// TIA Portal V20 export
FUNCTION_BLOCK "CallEquipment"   // FB177, LAD
TITLE = CallEquipment
// Template of an equipment module. This block contains the logic and futher calls (e.g. sequences, control modules, diagnostics etc.) of the equipment module.
// It can be used out of the box but also adapted to your own needs.
// stored: IsIECCheckEnabled true, MemoryReserve 100, Namespace Unit1.Em3, SetENOAutomatically true
   VAR_INPUT
      ZoneOperationEnable { ExternalWritable := 'False'} : "LWONIK_typeSafetyZoneManualOperation";
      unitEnableControlInterfaces { ExternalWritable := 'False'} : "LAF_typeEnableControlInterfaces";
      commandExcute { ExternalWritable := 'False'} : Bool;
   END_VAR
   VAR_IN_OUT
      unitStatus : "LAF_typeUnitStatus";   // Current unit status o be used in this EM
      emFeedback : "LUC_typeEmFeedback";   // Feedback of the EM to the Unit
      unitAlarmDB : "LAF_typeAlarms";   // Summarized EM Alarms for the Unit
   END_VAR
   VAR
      instSequenceWebGuid { ExternalWritable := 'False'} : "Unit1.Em3.Sequence_1_WebGuid";
      instWebGuidInitializedJob1 { ExternalWritable := 'False'} : "LAF_SelectJob";
      instWebGuidMotionCalculateJob2 { ExternalWritable := 'False'} : "LAF_SelectJob";
      instWebGuidMotionOneCellJob3 { ExternalWritable := 'False'} : "LAF_SelectJob";
      instWebGuidMotionFullStepJob4 { ExternalWritable := 'False'} : "LAF_SelectJob";
      instWebGuidMotionAutoJob5 { ExternalWritable := 'False'} : "LAF_SelectJob";
      instWebGuidMotionSemiStepJob6 { ExternalWritable := 'False'} : "LAF_SelectJob";
      instWebGuidMotionCycleStopJob7 { ExternalWritable := 'False'} : "LAF_SelectJob";
      instWebGuidMotionFastStopJob8 { ExternalWritable := 'False'} : "LAF_SelectJob";
      instCmMasterVirtualAxis { ExternalWritable := 'False'} : "LBC_AxisControl_TecPlcCn";
      instCmUnwinderVirtualAxis { ExternalWritable := 'False'} : "LBC_AxisControl_TecPlcCn";
      instCmDancerRegulatorOnOff { ExternalWritable := 'False'} : "LBC_TwoWayActuatorCn";
      instCmDancerSafetyPinIdlePosition { ExternalWritable := 'False'} : "LBC_DigitalSignalCn";
      instCmDancerEncoderAnalogInput { ExternalWritable := 'False'} : "LBC_AnalogInputCn";
      instCmLoadCellAnalogInput { ExternalWritable := 'False'} : "LBC_AnalogInputCn";
      instCmDancerElectroPneumaticRegulatorAnalogOutput { ExternalWritable := 'False'} : "LBC_AnalogOutputCn";
      instCmWebGuideEpc { ExternalWritable := 'False'} : "LER_EPC_CON600";
      instCmMasterAxisControlInterlockSummary { ExternalWritable := 'False'} : "LER_AxisControl_InterlockSummary";
      instCmUnwinderAxisControlInterlockSummary { ExternalWritable := 'False'} : "LER_AxisControl_InterlockSummary";
      statUnitStatus { ExternalWritable := 'False'} : "LAF_typeUnitStatus";   // Unit Status used in this EM
      instManageAlarms { ExternalWritable := 'False'} : "LAF_ManageAlarms";
      instEventsPFE { S7_SetPoint := 'True'} : "Unit1.Em3.EventsPFE";
      statLoadcellBuf { ExternalWritable := 'False'} : Int;
      statEnableManualCmds { ExternalWritable := 'False'} : Bool;
      statPulse { ExternalWritable := 'False'} : Array[0..99] of Bool;
      statTonTimer { ExternalWritable := 'False'} : Array[0..99] of TON_TIME;
      statTofTimer { ExternalWritable := 'False'} : Array[0..99] of TOF_TIME;
      instCheckCamRecipeChanged { ExternalWritable := 'False'} : "LER_CheckCamRecipeChanged";
      statCheckCamRecipeChangedStatus { ExternalWritable := 'False'} : Struct
         ValidParameters : Bool;
         ParameterChanged : Bool;
         ExecuteRequired : Bool;
      END_STRUCT;
      NGConveyorFull { ExternalVisible := 'False'; ExternalWritable := 'False'} : Bool;
      Stack1ConveyorFull { ExternalVisible := 'False'; ExternalWritable := 'False'} : Bool;
      Stack2ConveyorFull { ExternalVisible := 'False'; ExternalWritable := 'False'} : Bool;
      All_Full { ExternalVisible := 'False'; ExternalWritable := 'False'} : Bool;
      Stack1_Full_Abnormal { ExternalVisible := 'False'; ExternalWritable := 'False'} : Bool;
      Stack2_Full_Abnormal { ExternalVisible := 'False'; ExternalWritable := 'False'} : Bool;
      CutConveyorFull { ExternalVisible := 'False'; ExternalWritable := 'False'} : Bool;
      "Stack#1BA030Unuse" { ExternalVisible := 'False'; ExternalWritable := 'False'} : Bool;
      "Stack#2BA040Unuse" { ExternalVisible := 'False'; ExternalWritable := 'False'} : Bool;
      instCVFullChargeCheckCMD { S7_SetPoint := 'True'} : "LAF_SelectJob";
      CellCountDiv1 { S7_SetPoint := 'True'} : LReal;
      CellCountDiv2 { S7_SetPoint := 'True'} : LReal;
   END_VAR
   VAR_TEMP
      tempScInProduction : Bool;   // Mode Production and StateComplete
      tempScNoProduction : Bool;   // Mode Manual and StateComplete
   END_VAR
   VAR CONSTANT
      TO_DO_INSERT_PRECONDITIONS_HERE : Bool := TRUE;   // Template : Add em specific conditions here
      NO_JOB : DInt;   // No job
      TRUE : Bool := TRUE;
      FALSE : Bool := FALSE;
   END_VAR
   VAR_TEMP   // added for the SCL form of the ladder/FBD networks
      _w1 : Bool;
      _w2 : Bool;
   END_VAR
BEGIN

REGION Network 1: BLOCK INFO HEADER
   // (company) / (C) Copyright (year)
   // ---------------------------------------------------------------------------------
   // Title:                             (Title of this block)
   // Comment/Function: (that is implemented in the block)
   // Library/Family:           (that the source is dedicated to)
   // Author:                        (department / person in charge / contact)
   // Target System:          (test system with FW version)
   // Engineering:              TIA Portal (SW version)
   // Restrictions:               (OB types, etc.)
   // Requirements:           (hardware, technological package, etc.)
   // ---------------------------------------------------------------------------------
   // Change log table:
   // Version          | Date             | Signature      | Expert in charge  | Changes applied ------------------------|----------------------|-------------------------|--------------------------------|-----------------------
   // 001.000.000 | yyyy-mm-dd | 0x00000000 | (name of expert) | First released version
END_REGION

REGION Network 2: DESCRIPTION
   // This is a template block provided by the Automation Framework. It can be used to create an own project.
   // The Block Info Header is prepared to put in your own data.
   // Description of the block could be added here and the docu created by Code2Docu.
END_REGION

REGION Network 3: ******************** Equipment Control ********************
END_REGION

REGION Network 4: Interlink EM to Unit
   // This block links and unlinks the EM from the unit. The command to link/unlink can be set directly by the inputs of the block (e.g. to link/unlink based on any program logic) or through the InOut "hmiInterface". The block changes the output "isLinked" to true/false, depending on the command and if a change is allowed. A changed is allowed if the unit is in state aborted, clearing or stopped. The output "isLinked" is send back to the unit. If the EM is not linked, the unit ignores this EM.
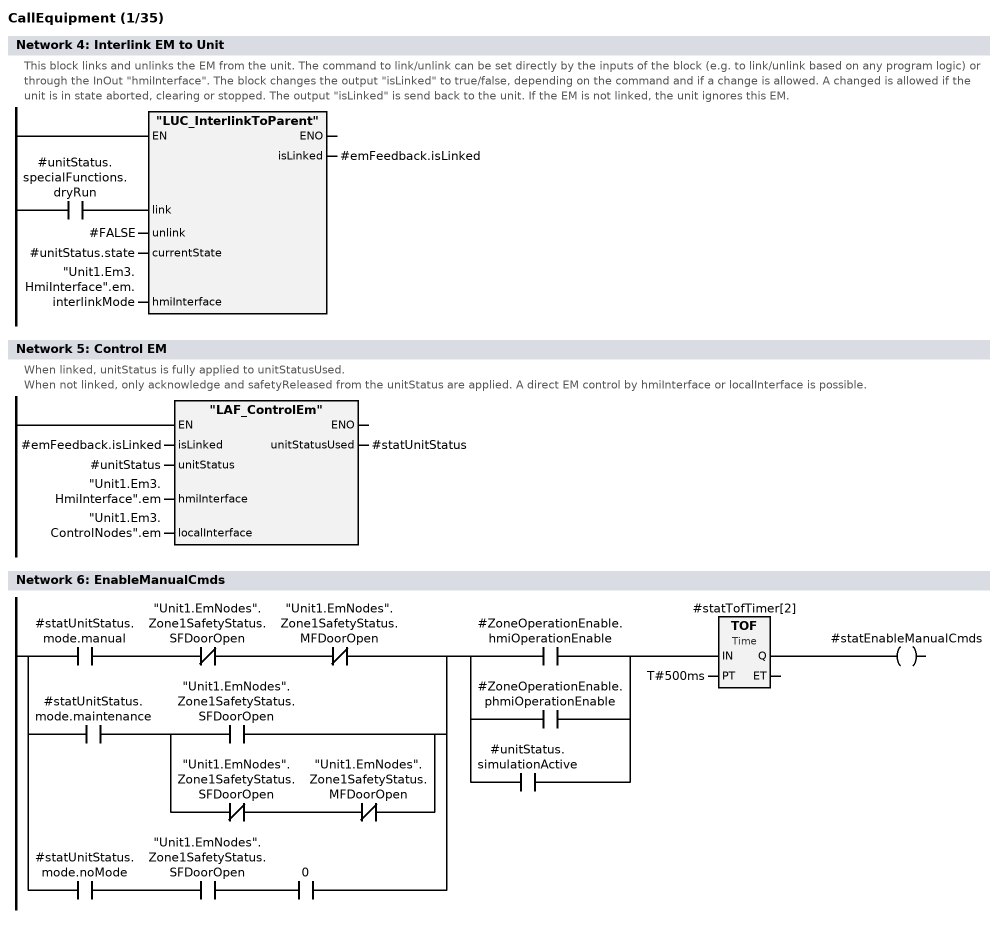
   RUNG wire#powerrail
      "LUC_InterlinkToParent"(link := wire#w1, unlink := #FALSE, currentState := #unitStatus.state, hmiInterface := "Unit1.Em3.HmiInterface".em.interlinkMode, isLinked => #emFeedback.isLinked)
   END_RUNG
   RUNG wire#powerrail
      Contact( #unitStatus.specialFunctions.dryRun )
   END_RUNG wire#w1
   // the same network as SCL:
   "LUC_InterlinkToParent"(link := #unitStatus.specialFunctions.dryRun,
                           unlink := #FALSE,
                           currentState := #unitStatus.state,
                           hmiInterface := "Unit1.Em3.HmiInterface".em.interlinkMode,
                           isLinked => #emFeedback.isLinked);
END_REGION

REGION Network 5: Control EM
   // When linked, unitStatus is fully applied to unitStatusUsed.
   // When not linked, only acknowledge and safetyReleased from the unitStatus are applied. A direct EM control by hmiInterface or localInterface is possible.
   RUNG wire#powerrail
      "LAF_ControlEm"(isLinked := #emFeedback.isLinked, unitStatus := #unitStatus, hmiInterface := "Unit1.Em3.HmiInterface".em, localInterface := "Unit1.Em3.ControlNodes".em, unitStatusUsed => #statUnitStatus)
   END_RUNG
   // the same network as SCL:
   "LAF_ControlEm"(isLinked := #emFeedback.isLinked,
                   unitStatus := #unitStatus,
                   hmiInterface := "Unit1.Em3.HmiInterface".em,
                   localInterface := "Unit1.Em3.ControlNodes".em,
                   unitStatusUsed => #statUnitStatus);
END_REGION

REGION Network 6: EnableManualCmds
   RUNG wire#powerrail
      Contact( #statUnitStatus.mode.manual )
      I_Contact( "Unit1.EmNodes".Zone1SafetyStatus.SFDoorOpen )
      I_Contact( "Unit1.EmNodes".Zone1SafetyStatus.MFDoorOpen )
      wire#w1
      Contact( #ZoneOperationEnable.hmiOperationEnable )
      wire#w3
      { S7_Templates := "time_type := Time" } #statTofTimer[2].TOF(pt := T#500ms, et =>)
      Coil( #statEnableManualCmds )
   END_RUNG
   RUNG wire#powerrail
      Contact( #statUnitStatus.mode.maintenance )
      wire#w2
      Contact( "Unit1.EmNodes".Zone1SafetyStatus.SFDoorOpen )
   END_RUNG wire#w1
   RUNG wire#w2
      I_Contact( "Unit1.EmNodes".Zone1SafetyStatus.SFDoorOpen )
      I_Contact( "Unit1.EmNodes".Zone1SafetyStatus.MFDoorOpen )
   END_RUNG wire#w1
   RUNG wire#powerrail
      Contact( #statUnitStatus.mode.noMode )
      Contact( "Unit1.EmNodes".Zone1SafetyStatus.SFDoorOpen )
      Contact( 0 )
   END_RUNG wire#w1
   RUNG wire#w1
      Contact( #ZoneOperationEnable.phmiOperationEnable )
   END_RUNG wire#w3
   RUNG wire#w1
      Contact( #unitStatus.simulationActive )
   END_RUNG wire#w3
   // the same network as SCL:
   #statTofTimer[2].TOF(IN := ((#statUnitStatus.mode.manual AND NOT "Unit1.EmNodes".Zone1SafetyStatus.SFDoorOpen AND NOT "Unit1.EmNodes".Zone1SafetyStatus.MFDoorOpen) OR (#statUnitStatus.mode.maintenance AND ("Unit1.EmNodes".Zone1SafetyStatus.SFDoorOpen OR (NOT "Unit1.EmNodes".Zone1SafetyStatus.SFDoorOpen AND NOT "Unit1.EmNodes".Zone1SafetyStatus.MFDoorOpen))) OR (#statUnitStatus.mode.noMode AND "Unit1.EmNodes".Zone1SafetyStatus.SFDoorOpen AND 0)) AND (#ZoneOperationEnable.hmiOperationEnable OR #ZoneOperationEnable.phmiOperationEnable OR #unitStatus.simulationActive),
                        PT := T#500ms);
   #statEnableManualCmds := #statTofTimer[2].Q;
END_REGION

REGION Network 7: Alarms Disabled
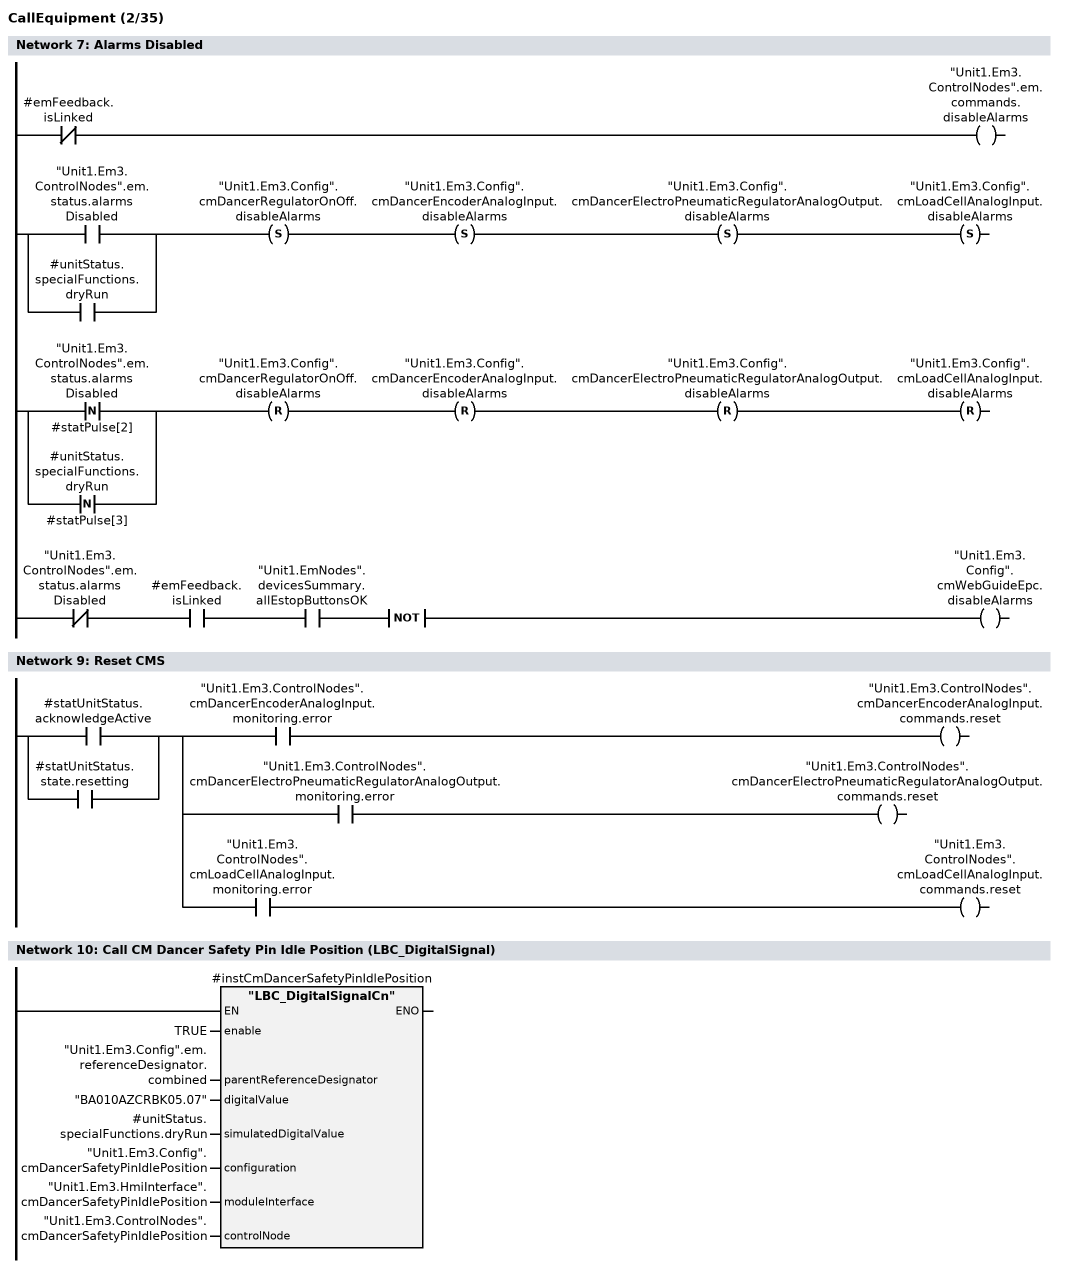
   RUNG wire#powerrail
      I_Contact( #emFeedback.isLinked )
      Coil( "Unit1.Em3.ControlNodes".em.commands.disableAlarms )
   END_RUNG
   RUNG wire#powerrail
      Contact( "Unit1.Em3.ControlNodes".em.status.alarmsDisabled )
      wire#w1
      S_Coil( "Unit1.Em3.Config".cmDancerRegulatorOnOff.disableAlarms )
      S_Coil( "Unit1.Em3.Config".cmDancerEncoderAnalogInput.disableAlarms )
      S_Coil( "Unit1.Em3.Config".cmDancerElectroPneumaticRegulatorAnalogOutput.disableAlarms )
      S_Coil( "Unit1.Em3.Config".cmLoadCellAnalogInput.disableAlarms )
   END_RUNG
   RUNG wire#powerrail
      Contact( #unitStatus.specialFunctions.dryRun )
   END_RUNG wire#w1
   RUNG wire#powerrail
      N_Contact(operand := "Unit1.Em3.ControlNodes".em.status.alarmsDisabled, bit := #statPulse[2])
      wire#w2
      R_Coil( "Unit1.Em3.Config".cmDancerRegulatorOnOff.disableAlarms )
      R_Coil( "Unit1.Em3.Config".cmDancerEncoderAnalogInput.disableAlarms )
      R_Coil( "Unit1.Em3.Config".cmDancerElectroPneumaticRegulatorAnalogOutput.disableAlarms )
      R_Coil( "Unit1.Em3.Config".cmLoadCellAnalogInput.disableAlarms )
   END_RUNG
   RUNG wire#powerrail
      N_Contact(operand := #unitStatus.specialFunctions.dryRun, bit := #statPulse[3])
   END_RUNG wire#w2
   RUNG wire#powerrail
      I_Contact( "Unit1.Em3.ControlNodes".em.status.alarmsDisabled )
      Contact( #emFeedback.isLinked )
      Contact( "Unit1.EmNodes".devicesSummary.allEstopButtonsOK )
      Not()
      Coil( "Unit1.Em3.Config".cmWebGuideEpc.disableAlarms )
   END_RUNG
   // the same network as SCL:
   "Unit1.Em3.ControlNodes".em.commands.disableAlarms := NOT #emFeedback.isLinked;
   IF "Unit1.Em3.ControlNodes".em.status.alarmsDisabled OR #unitStatus.specialFunctions.dryRun THEN
       "Unit1.Em3.Config".cmDancerRegulatorOnOff.disableAlarms := TRUE;
       "Unit1.Em3.Config".cmDancerEncoderAnalogInput.disableAlarms := TRUE;
       "Unit1.Em3.Config".cmDancerElectroPneumaticRegulatorAnalogOutput.disableAlarms := TRUE;
       "Unit1.Em3.Config".cmLoadCellAnalogInput.disableAlarms := TRUE;
   END_IF;
   #_w1 := NOT "Unit1.Em3.ControlNodes".em.status.alarmsDisabled AND #statPulse[2];   // falling edge of "Unit1.Em3.ControlNodes".em.status.alarmsDisabled
   #statPulse[2] := "Unit1.Em3.ControlNodes".em.status.alarmsDisabled;
   #_w2 := NOT #unitStatus.specialFunctions.dryRun AND #statPulse[3];   // falling edge of #unitStatus.specialFunctions.dryRun
   #statPulse[3] := #unitStatus.specialFunctions.dryRun;
   IF #_w1 OR #_w2 THEN
       "Unit1.Em3.Config".cmDancerRegulatorOnOff.disableAlarms := FALSE;
       "Unit1.Em3.Config".cmDancerEncoderAnalogInput.disableAlarms := FALSE;
       "Unit1.Em3.Config".cmDancerElectroPneumaticRegulatorAnalogOutput.disableAlarms := FALSE;
       "Unit1.Em3.Config".cmLoadCellAnalogInput.disableAlarms := FALSE;
   END_IF;
   "Unit1.Em3.Config".cmWebGuideEpc.disableAlarms := NOT (NOT "Unit1.Em3.ControlNodes".em.status.alarmsDisabled AND #emFeedback.isLinked AND "Unit1.EmNodes".devicesSummary.allEstopButtonsOK);
END_REGION

REGION Network 8: ******************** Control Modules (Sensors) ********************
   // Call control modules that are sensors before the em logic (jobs and sequence), so that the latest value is used in the logic.
END_REGION

REGION Network 9: Reset CMS
   RUNG wire#powerrail
      Contact( #statUnitStatus.acknowledgeActive )
      wire#w1
      Contact( "Unit1.Em3.ControlNodes".cmDancerEncoderAnalogInput.monitoring.error )
      Coil( "Unit1.Em3.ControlNodes".cmDancerEncoderAnalogInput.commands.reset )
   END_RUNG
   RUNG wire#powerrail
      Contact( #statUnitStatus.state.resetting )
   END_RUNG wire#w1
   RUNG wire#w1
      Contact( "Unit1.Em3.ControlNodes".cmDancerElectroPneumaticRegulatorAnalogOutput.monitoring.error )
      Coil( "Unit1.Em3.ControlNodes".cmDancerElectroPneumaticRegulatorAnalogOutput.commands.reset )
   END_RUNG
   RUNG wire#w1
      Contact( "Unit1.Em3.ControlNodes".cmLoadCellAnalogInput.monitoring.error )
      Coil( "Unit1.Em3.ControlNodes".cmLoadCellAnalogInput.commands.reset )
   END_RUNG
   // the same network as SCL:
   #_w1 := #statUnitStatus.acknowledgeActive OR #statUnitStatus.state.resetting;
   "Unit1.Em3.ControlNodes".cmDancerEncoderAnalogInput.commands.reset := #_w1 AND "Unit1.Em3.ControlNodes".cmDancerEncoderAnalogInput.monitoring.error;
   "Unit1.Em3.ControlNodes".cmDancerElectroPneumaticRegulatorAnalogOutput.commands.reset := #_w1 AND "Unit1.Em3.ControlNodes".cmDancerElectroPneumaticRegulatorAnalogOutput.monitoring.error;
   "Unit1.Em3.ControlNodes".cmLoadCellAnalogInput.commands.reset := #_w1 AND "Unit1.Em3.ControlNodes".cmLoadCellAnalogInput.monitoring.error;
END_REGION

REGION Network 10: Call CM Dancer Safety Pin Idle Position (LBC_DigitalSignal)
   RUNG wire#powerrail
      #instCmDancerSafetyPinIdlePosition(enable := TRUE, parentReferenceDesignator := "Unit1.Em3.Config".em.referenceDesignator.combined, digitalValue := "BA010AZCRBK05.07", simulatedDigitalValue := #unitStatus.specialFunctions.dryRun, configuration := "Unit1.Em3.Config".cmDancerSafetyPinIdlePosition, moduleInterface := "Unit1.Em3.HmiInterface".cmDancerSafetyPinIdlePosition, controlNode := "Unit1.Em3.ControlNodes".cmDancerSafetyPinIdlePosition)
   END_RUNG
   // the same network as SCL:
   #instCmDancerSafetyPinIdlePosition(enable := TRUE,   // "LBC_DigitalSignalCn"
                           parentReferenceDesignator := "Unit1.Em3.Config".em.referenceDesignator.combined,
                           digitalValue := "BA010AZCRBK05.07",
                           simulatedDigitalValue := #unitStatus.specialFunctions.dryRun,
                           configuration := "Unit1.Em3.Config".cmDancerSafetyPinIdlePosition,
                           moduleInterface := "Unit1.Em3.HmiInterface".cmDancerSafetyPinIdlePosition,
                           controlNode := "Unit1.Em3.ControlNodes".cmDancerSafetyPinIdlePosition);
END_REGION

REGION Network 11: Call CM Load Cell (LBC_AnalogInput)
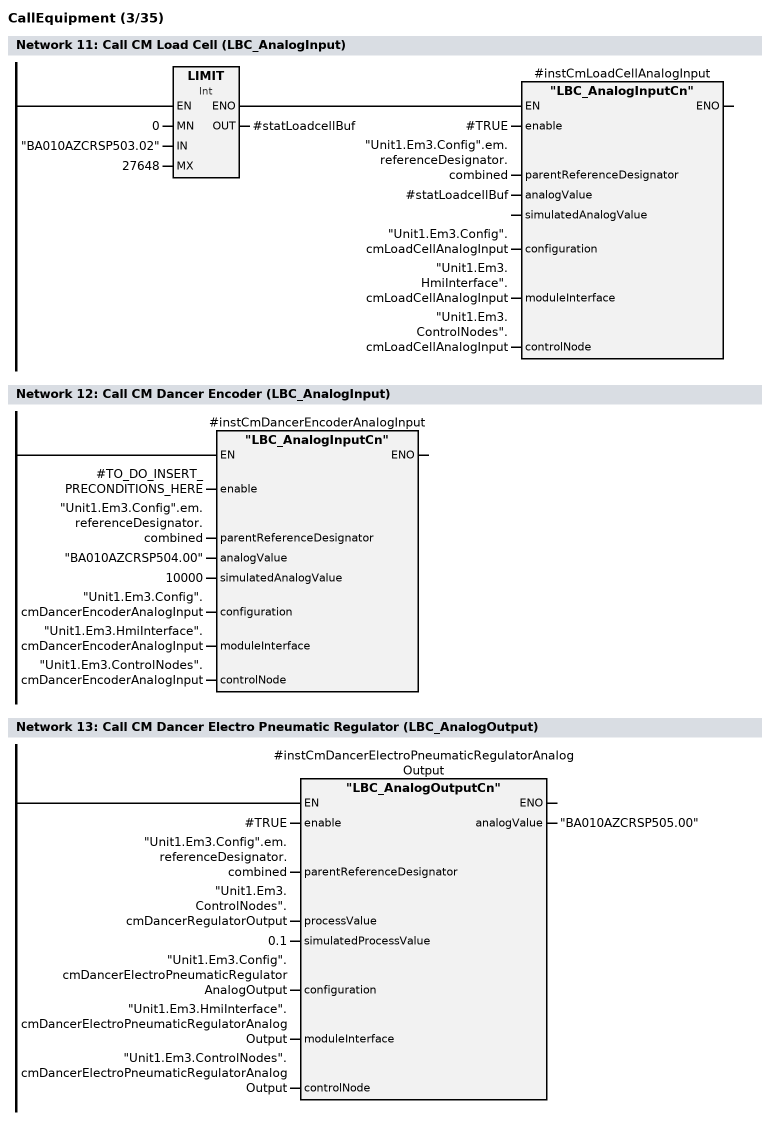
   RUNG wire#powerrail
      { S7_Templates := "value_type := Int" } Limit(mn := 0, in := "BA010AZCRSP503.02", mx := 27648, out => #statLoadcellBuf)
      #instCmLoadCellAnalogInput(enable := #TRUE, parentReferenceDesignator := "Unit1.Em3.Config".em.referenceDesignator.combined, analogValue := #statLoadcellBuf, simulatedAnalogValue :=, configuration := "Unit1.Em3.Config".cmLoadCellAnalogInput, moduleInterface := "Unit1.Em3.HmiInterface".cmLoadCellAnalogInput, controlNode := "Unit1.Em3.ControlNodes".cmLoadCellAnalogInput)
   END_RUNG
   // the same network as SCL:
   #statLoadcellBuf := LIMIT(MN := 0, IN := "BA010AZCRSP503.02", MX := 27648);
   #instCmLoadCellAnalogInput(enable := #TRUE,   // "LBC_AnalogInputCn"
                           parentReferenceDesignator := "Unit1.Em3.Config".em.referenceDesignator.combined,
                           analogValue := #statLoadcellBuf,
                           configuration := "Unit1.Em3.Config".cmLoadCellAnalogInput,
                           moduleInterface := "Unit1.Em3.HmiInterface".cmLoadCellAnalogInput,
                           controlNode := "Unit1.Em3.ControlNodes".cmLoadCellAnalogInput);
END_REGION

REGION Network 12: Call CM Dancer Encoder (LBC_AnalogInput)
   RUNG wire#powerrail
      #instCmDancerEncoderAnalogInput(enable := #TO_DO_INSERT_PRECONDITIONS_HERE, parentReferenceDesignator := "Unit1.Em3.Config".em.referenceDesignator.combined, analogValue := "BA010AZCRSP504.00", simulatedAnalogValue := 10000, configuration := "Unit1.Em3.Config".cmDancerEncoderAnalogInput, moduleInterface := "Unit1.Em3.HmiInterface".cmDancerEncoderAnalogInput, controlNode := "Unit1.Em3.ControlNodes".cmDancerEncoderAnalogInput)
   END_RUNG
   // the same network as SCL:
   #instCmDancerEncoderAnalogInput(enable := #TO_DO_INSERT_PRECONDITIONS_HERE,   // "LBC_AnalogInputCn"
                           parentReferenceDesignator := "Unit1.Em3.Config".em.referenceDesignator.combined,
                           analogValue := "BA010AZCRSP504.00",
                           simulatedAnalogValue := 10000,
                           configuration := "Unit1.Em3.Config".cmDancerEncoderAnalogInput,
                           moduleInterface := "Unit1.Em3.HmiInterface".cmDancerEncoderAnalogInput,
                           controlNode := "Unit1.Em3.ControlNodes".cmDancerEncoderAnalogInput);
END_REGION

REGION Network 13: Call CM Dancer Electro Pneumatic Regulator (LBC_AnalogOutput)
   RUNG wire#powerrail
      #instCmDancerElectroPneumaticRegulatorAnalogOutput(enable := #TRUE, parentReferenceDesignator := "Unit1.Em3.Config".em.referenceDesignator.combined, processValue := "Unit1.Em3.ControlNodes".cmDancerRegulatorOutput, simulatedProcessValue := 0.1, configuration := "Unit1.Em3.Config".cmDancerElectroPneumaticRegulatorAnalogOutput, moduleInterface := "Unit1.Em3.HmiInterface".cmDancerElectroPneumaticRegulatorAnalogOutput, controlNode := "Unit1.Em3.ControlNodes".cmDancerElectroPneumaticRegulatorAnalogOutput, analogValue => "BA010AZCRSP505.00")
   END_RUNG
   // the same network as SCL:
   #instCmDancerElectroPneumaticRegulatorAnalogOutput(enable := #TRUE,   // "LBC_AnalogOutputCn"
                           parentReferenceDesignator := "Unit1.Em3.Config".em.referenceDesignator.combined,
                           processValue := "Unit1.Em3.ControlNodes".cmDancerRegulatorOutput,
                           simulatedProcessValue := 0.1,
                           configuration := "Unit1.Em3.Config".cmDancerElectroPneumaticRegulatorAnalogOutput,
                           moduleInterface := "Unit1.Em3.HmiInterface".cmDancerElectroPneumaticRegulatorAnalogOutput,
                           controlNode := "Unit1.Em3.ControlNodes".cmDancerElectroPneumaticRegulatorAnalogOutput,
                           analogValue => "BA010AZCRSP505.00");
END_REGION

REGION Network 14: ******************** Equipment Logic ********************
END_REGION

REGION Network 15: Map Unit Status to Sequence Status [1] WebGuid
   // This block maps the unit status to the seuqnce status. Thus, it controls the sequence depending on the unit status. E.g. it sets the sequence to automatic when the unit state is in productions. This blocks work perfectly with the sequences provided in the AF. 
   // This typed block (MapUnitStatusToSequence) could be adjusted to specific application requirements or if other, user-defined sequences are used.
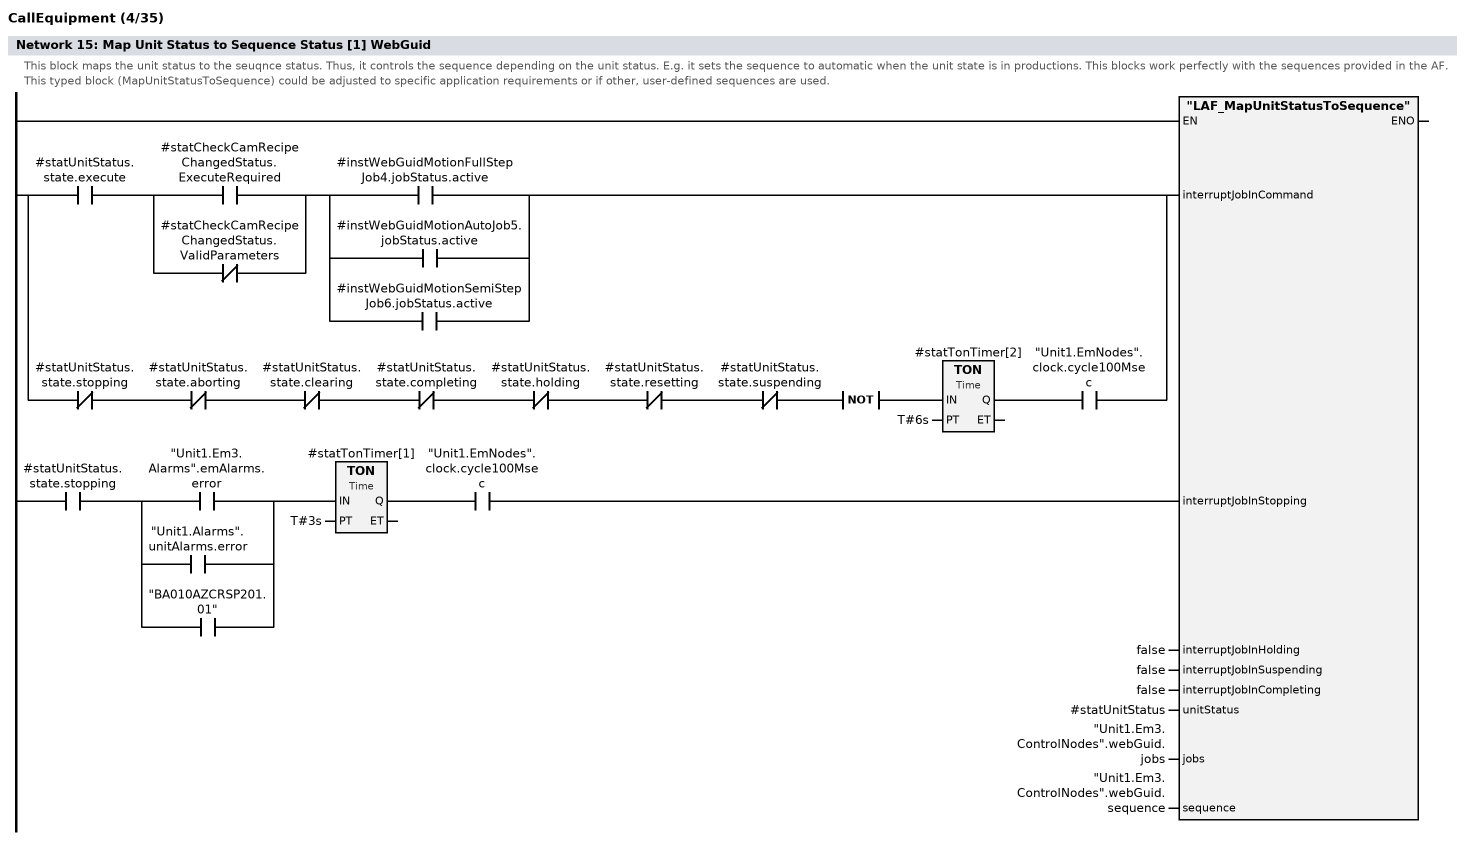
   RUNG wire#powerrail
      "LAF_MapUnitStatusToSequence"(interruptJobInCommand := wire#w3, interruptJobInStopping := wire#w6, interruptJobInHolding := false, interruptJobInSuspending := false, interruptJobInCompleting := false, unitStatus := #statUnitStatus, jobs := "Unit1.Em3.ControlNodes".webGuid.jobs, sequence := "Unit1.Em3.ControlNodes".webGuid.sequence)
   END_RUNG
   RUNG wire#powerrail
      Contact( #statUnitStatus.state.execute )
      wire#w1
      Contact( #statCheckCamRecipeChangedStatus.ExecuteRequired )
      wire#w2
      Contact( #instWebGuidMotionFullStepJob4.jobStatus.active )
   END_RUNG wire#w3
   RUNG wire#w1
      I_Contact( #statCheckCamRecipeChangedStatus.ValidParameters )
   END_RUNG wire#w2
   RUNG wire#w2
      Contact( #instWebGuidMotionAutoJob5.jobStatus.active )
   END_RUNG wire#w3
   RUNG wire#w2
      Contact( #instWebGuidMotionSemiStepJob6.jobStatus.active )
   END_RUNG wire#w3
   RUNG wire#powerrail
      I_Contact( #statUnitStatus.state.stopping )
      I_Contact( #statUnitStatus.state.aborting )
      I_Contact( #statUnitStatus.state.clearing )
      I_Contact( #statUnitStatus.state.completing )
      I_Contact( #statUnitStatus.state.holding )
      I_Contact( #statUnitStatus.state.resetting )
      I_Contact( #statUnitStatus.state.suspending )
      Not()
      { S7_Templates := "time_type := Time" } #statTonTimer[2].TON(pt := T#6s, et =>)
      Contact( "Unit1.EmNodes".clock.cycle100Msec )
   END_RUNG wire#w3
   RUNG wire#powerrail
      Contact( #statUnitStatus.state.stopping )
      wire#w4
      Contact( "Unit1.Em3.Alarms".emAlarms.error )
      wire#w5
      { S7_Templates := "time_type := Time" } #statTonTimer[1].TON(pt := T#3s, et =>)
      Contact( "Unit1.EmNodes".clock.cycle100Msec )
   END_RUNG wire#w6
   RUNG wire#w4
      Contact( "Unit1.Alarms".unitAlarms.error )
   END_RUNG wire#w5
   RUNG wire#w4
      Contact( "BA010AZCRSP201.01" )
   END_RUNG wire#w5
   // the same network as SCL:
   #statTonTimer[2].TON(IN := NOT (NOT #statUnitStatus.state.stopping AND NOT #statUnitStatus.state.aborting AND NOT #statUnitStatus.state.clearing AND NOT #statUnitStatus.state.completing AND NOT #statUnitStatus.state.holding AND NOT #statUnitStatus.state.resetting AND NOT #statUnitStatus.state.suspending),
                        PT := T#6s);
   #_w1 := (#statUnitStatus.state.execute AND (#statCheckCamRecipeChangedStatus.ExecuteRequired OR NOT #statCheckCamRecipeChangedStatus.ValidParameters) AND (#instWebGuidMotionFullStepJob4.jobStatus.active OR #instWebGuidMotionAutoJob5.jobStatus.active OR #instWebGuidMotionSemiStepJob6.jobStatus.active)) OR (#statTonTimer[2].Q AND "Unit1.EmNodes".clock.cycle100Msec);
   #statTonTimer[1].TON(IN := #statUnitStatus.state.stopping AND ("Unit1.Em3.Alarms".emAlarms.error OR "Unit1.Alarms".unitAlarms.error OR "BA010AZCRSP201.01"),
                        PT := T#3s);
   "LAF_MapUnitStatusToSequence"(interruptJobInCommand := #_w1,
                           interruptJobInStopping := #statTonTimer[1].Q AND "Unit1.EmNodes".clock.cycle100Msec,
                           interruptJobInHolding := false,
                           interruptJobInSuspending := false,
                           interruptJobInCompleting := false,
                           unitStatus := #statUnitStatus,
                           jobs := "Unit1.Em3.ControlNodes".webGuid.jobs,
                           sequence := "Unit1.Em3.ControlNodes".webGuid.sequence);
END_REGION

REGION Network 16: C/V Full Charge Check before motion job select
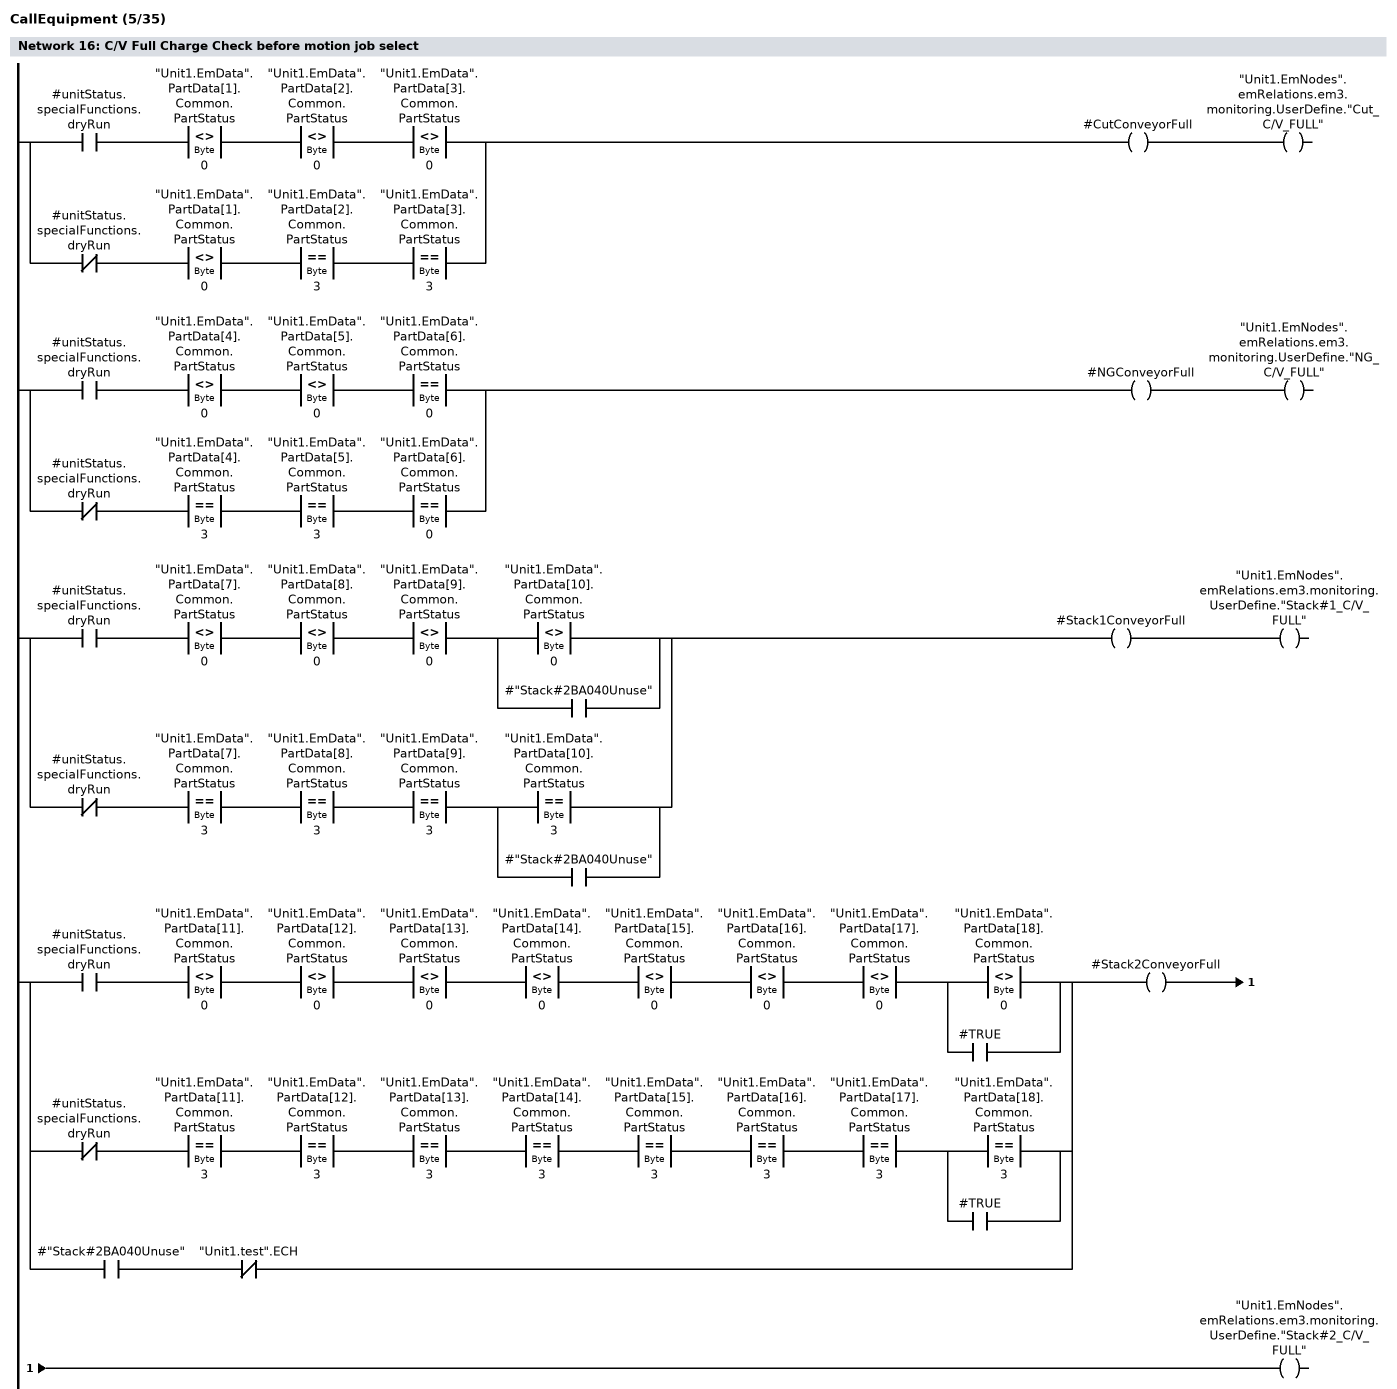
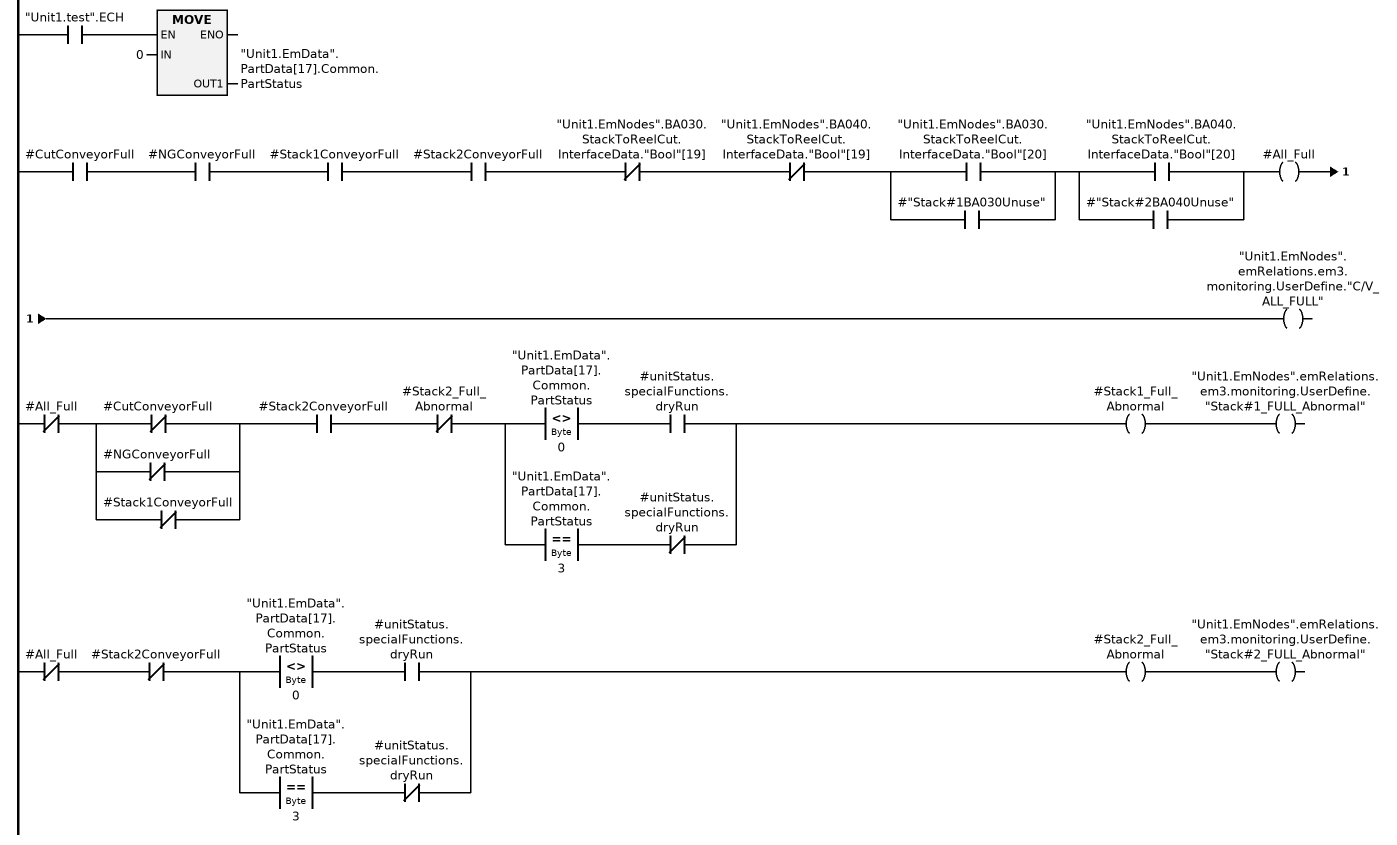
   RUNG wire#powerrail
      Contact( #unitStatus.specialFunctions.dryRun )
      { S7_Templates := "SrcType := Byte" } NE_Contact(in1 := "Unit1.EmData".PartData[1].Common.PartStatus, in2 := 0)
      { S7_Templates := "SrcType := Byte" } NE_Contact(in1 := "Unit1.EmData".PartData[2].Common.PartStatus, in2 := 0)
      { S7_Templates := "SrcType := Byte" } NE_Contact(in1 := "Unit1.EmData".PartData[3].Common.PartStatus, in2 := 0)
      wire#w1
      Coil( #CutConveyorFull )
      Coil( "Unit1.EmNodes".emRelations.em3.monitoring.UserDefine."Cut_C/V_FULL" )
   END_RUNG
   RUNG wire#powerrail
      I_Contact( #unitStatus.specialFunctions.dryRun )
      { S7_Templates := "SrcType := Byte" } NE_Contact(in1 := "Unit1.EmData".PartData[1].Common.PartStatus, in2 := 0)
      { S7_Templates := "SrcType := Byte" } EQ_Contact(in1 := "Unit1.EmData".PartData[2].Common.PartStatus, in2 := 3)
      { S7_Templates := "SrcType := Byte" } EQ_Contact(in1 := "Unit1.EmData".PartData[3].Common.PartStatus, in2 := 3)
   END_RUNG wire#w1
   RUNG wire#powerrail
      Contact( #unitStatus.specialFunctions.dryRun )
      { S7_Templates := "SrcType := Byte" } NE_Contact(in1 := "Unit1.EmData".PartData[4].Common.PartStatus, in2 := 0)
      { S7_Templates := "SrcType := Byte" } NE_Contact(in1 := "Unit1.EmData".PartData[5].Common.PartStatus, in2 := 0)
      { S7_Templates := "SrcType := Byte" } EQ_Contact(in1 := "Unit1.EmData".PartData[6].Common.PartStatus, in2 := 0)
      wire#w2
      Coil( #NGConveyorFull )
      Coil( "Unit1.EmNodes".emRelations.em3.monitoring.UserDefine."NG_C/V_FULL" )
   END_RUNG
   RUNG wire#powerrail
      I_Contact( #unitStatus.specialFunctions.dryRun )
      { S7_Templates := "SrcType := Byte" } EQ_Contact(in1 := "Unit1.EmData".PartData[4].Common.PartStatus, in2 := 3)
      { S7_Templates := "SrcType := Byte" } EQ_Contact(in1 := "Unit1.EmData".PartData[5].Common.PartStatus, in2 := 3)
      { S7_Templates := "SrcType := Byte" } EQ_Contact(in1 := "Unit1.EmData".PartData[6].Common.PartStatus, in2 := 0)
   END_RUNG wire#w2
   RUNG wire#powerrail
      Contact( #unitStatus.specialFunctions.dryRun )
      { S7_Templates := "SrcType := Byte" } NE_Contact(in1 := "Unit1.EmData".PartData[7].Common.PartStatus, in2 := 0)
      { S7_Templates := "SrcType := Byte" } NE_Contact(in1 := "Unit1.EmData".PartData[8].Common.PartStatus, in2 := 0)
      { S7_Templates := "SrcType := Byte" } NE_Contact(in1 := "Unit1.EmData".PartData[9].Common.PartStatus, in2 := 0)
      wire#w3
      { S7_Templates := "SrcType := Byte" } NE_Contact(in1 := "Unit1.EmData".PartData[10].Common.PartStatus, in2 := 0)
      wire#w4
      Coil( #Stack1ConveyorFull )
      Coil( "Unit1.EmNodes".emRelations.em3.monitoring.UserDefine."Stack#1_C/V_FULL" )
   END_RUNG
   RUNG wire#w3
      Contact( #"Stack#2BA040Unuse" )
   END_RUNG wire#w4
   RUNG wire#powerrail
      I_Contact( #unitStatus.specialFunctions.dryRun )
      { S7_Templates := "SrcType := Byte" } EQ_Contact(in1 := "Unit1.EmData".PartData[7].Common.PartStatus, in2 := 3)
      { S7_Templates := "SrcType := Byte" } EQ_Contact(in1 := "Unit1.EmData".PartData[8].Common.PartStatus, in2 := 3)
      { S7_Templates := "SrcType := Byte" } EQ_Contact(in1 := "Unit1.EmData".PartData[9].Common.PartStatus, in2 := 3)
      wire#w5
      { S7_Templates := "SrcType := Byte" } EQ_Contact(in1 := "Unit1.EmData".PartData[10].Common.PartStatus, in2 := 3)
   END_RUNG wire#w4
   RUNG wire#w5
      Contact( #"Stack#2BA040Unuse" )
   END_RUNG wire#w4
   RUNG wire#powerrail
      Contact( #unitStatus.specialFunctions.dryRun )
      { S7_Templates := "SrcType := Byte" } NE_Contact(in1 := "Unit1.EmData".PartData[11].Common.PartStatus, in2 := 0)
      { S7_Templates := "SrcType := Byte" } NE_Contact(in1 := "Unit1.EmData".PartData[12].Common.PartStatus, in2 := 0)
      { S7_Templates := "SrcType := Byte" } NE_Contact(in1 := "Unit1.EmData".PartData[13].Common.PartStatus, in2 := 0)
      { S7_Templates := "SrcType := Byte" } NE_Contact(in1 := "Unit1.EmData".PartData[14].Common.PartStatus, in2 := 0)
      { S7_Templates := "SrcType := Byte" } NE_Contact(in1 := "Unit1.EmData".PartData[15].Common.PartStatus, in2 := 0)
      { S7_Templates := "SrcType := Byte" } NE_Contact(in1 := "Unit1.EmData".PartData[16].Common.PartStatus, in2 := 0)
      { S7_Templates := "SrcType := Byte" } NE_Contact(in1 := "Unit1.EmData".PartData[17].Common.PartStatus, in2 := 0)
      wire#w6
      { S7_Templates := "SrcType := Byte" } NE_Contact(in1 := "Unit1.EmData".PartData[18].Common.PartStatus, in2 := 0)
      wire#w7
      Coil( #Stack2ConveyorFull )
      Coil( "Unit1.EmNodes".emRelations.em3.monitoring.UserDefine."Stack#2_C/V_FULL" )
   END_RUNG
   RUNG wire#w6
      Contact( #TRUE )
   END_RUNG wire#w7
   RUNG wire#powerrail
      I_Contact( #unitStatus.specialFunctions.dryRun )
      { S7_Templates := "SrcType := Byte" } EQ_Contact(in1 := "Unit1.EmData".PartData[11].Common.PartStatus, in2 := 3)
      { S7_Templates := "SrcType := Byte" } EQ_Contact(in1 := "Unit1.EmData".PartData[12].Common.PartStatus, in2 := 3)
      { S7_Templates := "SrcType := Byte" } EQ_Contact(in1 := "Unit1.EmData".PartData[13].Common.PartStatus, in2 := 3)
      { S7_Templates := "SrcType := Byte" } EQ_Contact(in1 := "Unit1.EmData".PartData[14].Common.PartStatus, in2 := 3)
      { S7_Templates := "SrcType := Byte" } EQ_Contact(in1 := "Unit1.EmData".PartData[15].Common.PartStatus, in2 := 3)
      { S7_Templates := "SrcType := Byte" } EQ_Contact(in1 := "Unit1.EmData".PartData[16].Common.PartStatus, in2 := 3)
      { S7_Templates := "SrcType := Byte" } EQ_Contact(in1 := "Unit1.EmData".PartData[17].Common.PartStatus, in2 := 3)
      wire#w8
      { S7_Templates := "SrcType := Byte" } EQ_Contact(in1 := "Unit1.EmData".PartData[18].Common.PartStatus, in2 := 3)
   END_RUNG wire#w7
   RUNG wire#w8
      Contact( #TRUE )
   END_RUNG wire#w7
   RUNG wire#powerrail
      Contact( #"Stack#2BA040Unuse" )
      I_Contact( "Unit1.test".ECH )
   END_RUNG wire#w7
   RUNG wire#powerrail
      Contact( "Unit1.test".ECH )
      Move(in := 0, out1 => "Unit1.EmData".PartData[17].Common.PartStatus)
   END_RUNG
   RUNG wire#powerrail
      Contact( #CutConveyorFull )
      Contact( #NGConveyorFull )
      Contact( #Stack1ConveyorFull )
      Contact( #Stack2ConveyorFull )
      I_Contact( "Unit1.EmNodes".BA030.StackToReelCut.InterfaceData."Bool"[19] )
      I_Contact( "Unit1.EmNodes".BA040.StackToReelCut.InterfaceData."Bool"[19] )
      wire#w9
      Contact( "Unit1.EmNodes".BA030.StackToReelCut.InterfaceData."Bool"[20] )
      wire#w10
      Contact( "Unit1.EmNodes".BA040.StackToReelCut.InterfaceData."Bool"[20] )
      wire#w11
      Coil( #All_Full )
      Coil( "Unit1.EmNodes".emRelations.em3.monitoring.UserDefine."C/V_ALL_FULL" )
   END_RUNG
   RUNG wire#w9
      Contact( #"Stack#1BA030Unuse" )
   END_RUNG wire#w10
   RUNG wire#w10
      Contact( #"Stack#2BA040Unuse" )
   END_RUNG wire#w11
   RUNG wire#powerrail
      I_Contact( #All_Full )
      wire#w12
      I_Contact( #CutConveyorFull )
      wire#w13
      Contact( #Stack2ConveyorFull )
      I_Contact( #Stack2_Full_Abnormal )
      wire#w14
      { S7_Templates := "SrcType := Byte" } NE_Contact(in1 := "Unit1.EmData".PartData[17].Common.PartStatus, in2 := 0)
      Contact( #unitStatus.specialFunctions.dryRun )
      wire#w15
      Coil( #Stack1_Full_Abnormal )
      Coil( "Unit1.EmNodes".emRelations.em3.monitoring.UserDefine."Stack#1_FULL_Abnormal" )
   END_RUNG
   RUNG wire#w12
      I_Contact( #NGConveyorFull )
   END_RUNG wire#w13
   RUNG wire#w12
      I_Contact( #Stack1ConveyorFull )
   END_RUNG wire#w13
   RUNG wire#w14
      { S7_Templates := "SrcType := Byte" } EQ_Contact(in1 := "Unit1.EmData".PartData[17].Common.PartStatus, in2 := 3)
      I_Contact( #unitStatus.specialFunctions.dryRun )
   END_RUNG wire#w15
   RUNG wire#powerrail
      I_Contact( #All_Full )
      I_Contact( #Stack2ConveyorFull )
      wire#w16
      { S7_Templates := "SrcType := Byte" } NE_Contact(in1 := "Unit1.EmData".PartData[17].Common.PartStatus, in2 := 0)
      Contact( #unitStatus.specialFunctions.dryRun )
      wire#w17
      Coil( #Stack2_Full_Abnormal )
      Coil( "Unit1.EmNodes".emRelations.em3.monitoring.UserDefine."Stack#2_FULL_Abnormal" )
   END_RUNG
   RUNG wire#w16
      { S7_Templates := "SrcType := Byte" } EQ_Contact(in1 := "Unit1.EmData".PartData[17].Common.PartStatus, in2 := 3)
      I_Contact( #unitStatus.specialFunctions.dryRun )
   END_RUNG wire#w17
   // the same network as SCL:
   #CutConveyorFull := (#unitStatus.specialFunctions.dryRun AND ("Unit1.EmData".PartData[1].Common.PartStatus <> 0) AND ("Unit1.EmData".PartData[2].Common.PartStatus <> 0) AND ("Unit1.EmData".PartData[3].Common.PartStatus <> 0)) OR (NOT #unitStatus.specialFunctions.dryRun AND ("Unit1.EmData".PartData[1].Common.PartStatus <> 0) AND ("Unit1.EmData".PartData[2].Common.PartStatus = 3) AND ("Unit1.EmData".PartData[3].Common.PartStatus = 3));
   "Unit1.EmNodes".emRelations.em3.monitoring.UserDefine."Cut_C/V_FULL" := #CutConveyorFull;
   #NGConveyorFull := (#unitStatus.specialFunctions.dryRun AND ("Unit1.EmData".PartData[4].Common.PartStatus <> 0) AND ("Unit1.EmData".PartData[5].Common.PartStatus <> 0) AND ("Unit1.EmData".PartData[6].Common.PartStatus = 0)) OR (NOT #unitStatus.specialFunctions.dryRun AND ("Unit1.EmData".PartData[4].Common.PartStatus = 3) AND ("Unit1.EmData".PartData[5].Common.PartStatus = 3) AND ("Unit1.EmData".PartData[6].Common.PartStatus = 0));
   "Unit1.EmNodes".emRelations.em3.monitoring.UserDefine."NG_C/V_FULL" := #NGConveyorFull;
   #Stack1ConveyorFull := (#unitStatus.specialFunctions.dryRun AND ("Unit1.EmData".PartData[7].Common.PartStatus <> 0) AND ("Unit1.EmData".PartData[8].Common.PartStatus <> 0) AND ("Unit1.EmData".PartData[9].Common.PartStatus <> 0) AND (("Unit1.EmData".PartData[10].Common.PartStatus <> 0) OR #"Stack#2BA040Unuse")) OR (NOT #unitStatus.specialFunctions.dryRun AND ("Unit1.EmData".PartData[7].Common.PartStatus = 3) AND ("Unit1.EmData".PartData[8].Common.PartStatus = 3) AND ("Unit1.EmData".PartData[9].Common.PartStatus = 3) AND (("Unit1.EmData".PartData[10].Common.PartStatus = 3) OR #"Stack#2BA040Unuse"));
   "Unit1.EmNodes".emRelations.em3.monitoring.UserDefine."Stack#1_C/V_FULL" := #Stack1ConveyorFull;
   #Stack2ConveyorFull := (#unitStatus.specialFunctions.dryRun AND ("Unit1.EmData".PartData[11].Common.PartStatus <> 0) AND ("Unit1.EmData".PartData[12].Common.PartStatus <> 0) AND ("Unit1.EmData".PartData[13].Common.PartStatus <> 0) AND ("Unit1.EmData".PartData[14].Common.PartStatus <> 0) AND ("Unit1.EmData".PartData[15].Common.PartStatus <> 0) AND ("Unit1.EmData".PartData[16].Common.PartStatus <> 0) AND ("Unit1.EmData".PartData[17].Common.PartStatus <> 0) AND (("Unit1.EmData".PartData[18].Common.PartStatus <> 0) OR #TRUE)) OR (NOT #unitStatus.specialFunctions.dryRun AND ("Unit1.EmData".PartData[11].Common.PartStatus = 3) AND ("Unit1.EmData".PartData[12].Common.PartStatus = 3) AND ("Unit1.EmData".PartData[13].Common.PartStatus = 3) AND ("Unit1.EmData".PartData[14].Common.PartStatus = 3) AND ("Unit1.EmData".PartData[15].Common.PartStatus = 3) AND ("Unit1.EmData".PartData[16].Common.PartStatus = 3) AND ("Unit1.EmData".PartData[17].Common.PartStatus = 3) AND (("Unit1.EmData".PartData[18].Common.PartStatus = 3) OR #TRUE)) OR (#"Stack#2BA040Unuse" AND NOT "Unit1.test".ECH);
   "Unit1.EmNodes".emRelations.em3.monitoring.UserDefine."Stack#2_C/V_FULL" := #Stack2ConveyorFull;
   IF "Unit1.test".ECH THEN "Unit1.EmData".PartData[17].Common.PartStatus := 0; END_IF;
   #All_Full := #CutConveyorFull AND #NGConveyorFull AND #Stack1ConveyorFull AND #Stack2ConveyorFull AND NOT "Unit1.EmNodes".BA030.StackToReelCut.InterfaceData."Bool"[19] AND NOT "Unit1.EmNodes".BA040.StackToReelCut.InterfaceData."Bool"[19] AND ("Unit1.EmNodes".BA030.StackToReelCut.InterfaceData."Bool"[20] OR #"Stack#1BA030Unuse") AND ("Unit1.EmNodes".BA040.StackToReelCut.InterfaceData."Bool"[20] OR #"Stack#2BA040Unuse");
   "Unit1.EmNodes".emRelations.em3.monitoring.UserDefine."C/V_ALL_FULL" := #All_Full;
   #Stack1_Full_Abnormal := NOT #All_Full AND (NOT #CutConveyorFull OR NOT #NGConveyorFull OR NOT #Stack1ConveyorFull) AND #Stack2ConveyorFull AND NOT #Stack2_Full_Abnormal AND ((("Unit1.EmData".PartData[17].Common.PartStatus <> 0) AND #unitStatus.specialFunctions.dryRun) OR (("Unit1.EmData".PartData[17].Common.PartStatus = 3) AND NOT #unitStatus.specialFunctions.dryRun));
   "Unit1.EmNodes".emRelations.em3.monitoring.UserDefine."Stack#1_FULL_Abnormal" := #Stack1_Full_Abnormal;
   #Stack2_Full_Abnormal := NOT #All_Full AND NOT #Stack2ConveyorFull AND ((("Unit1.EmData".PartData[17].Common.PartStatus <> 0) AND #unitStatus.specialFunctions.dryRun) OR (("Unit1.EmData".PartData[17].Common.PartStatus = 3) AND NOT #unitStatus.specialFunctions.dryRun));
   "Unit1.EmNodes".emRelations.em3.monitoring.UserDefine."Stack#2_FULL_Abnormal" := #Stack2_Full_Abnormal;
END_REGION

REGION Network 17: Select Job [1] Initialized
   // Decide which Step Sequence to start depending on the OMAC State and EM conditions
   // First Move Block is to Initialize the jobSelect Number
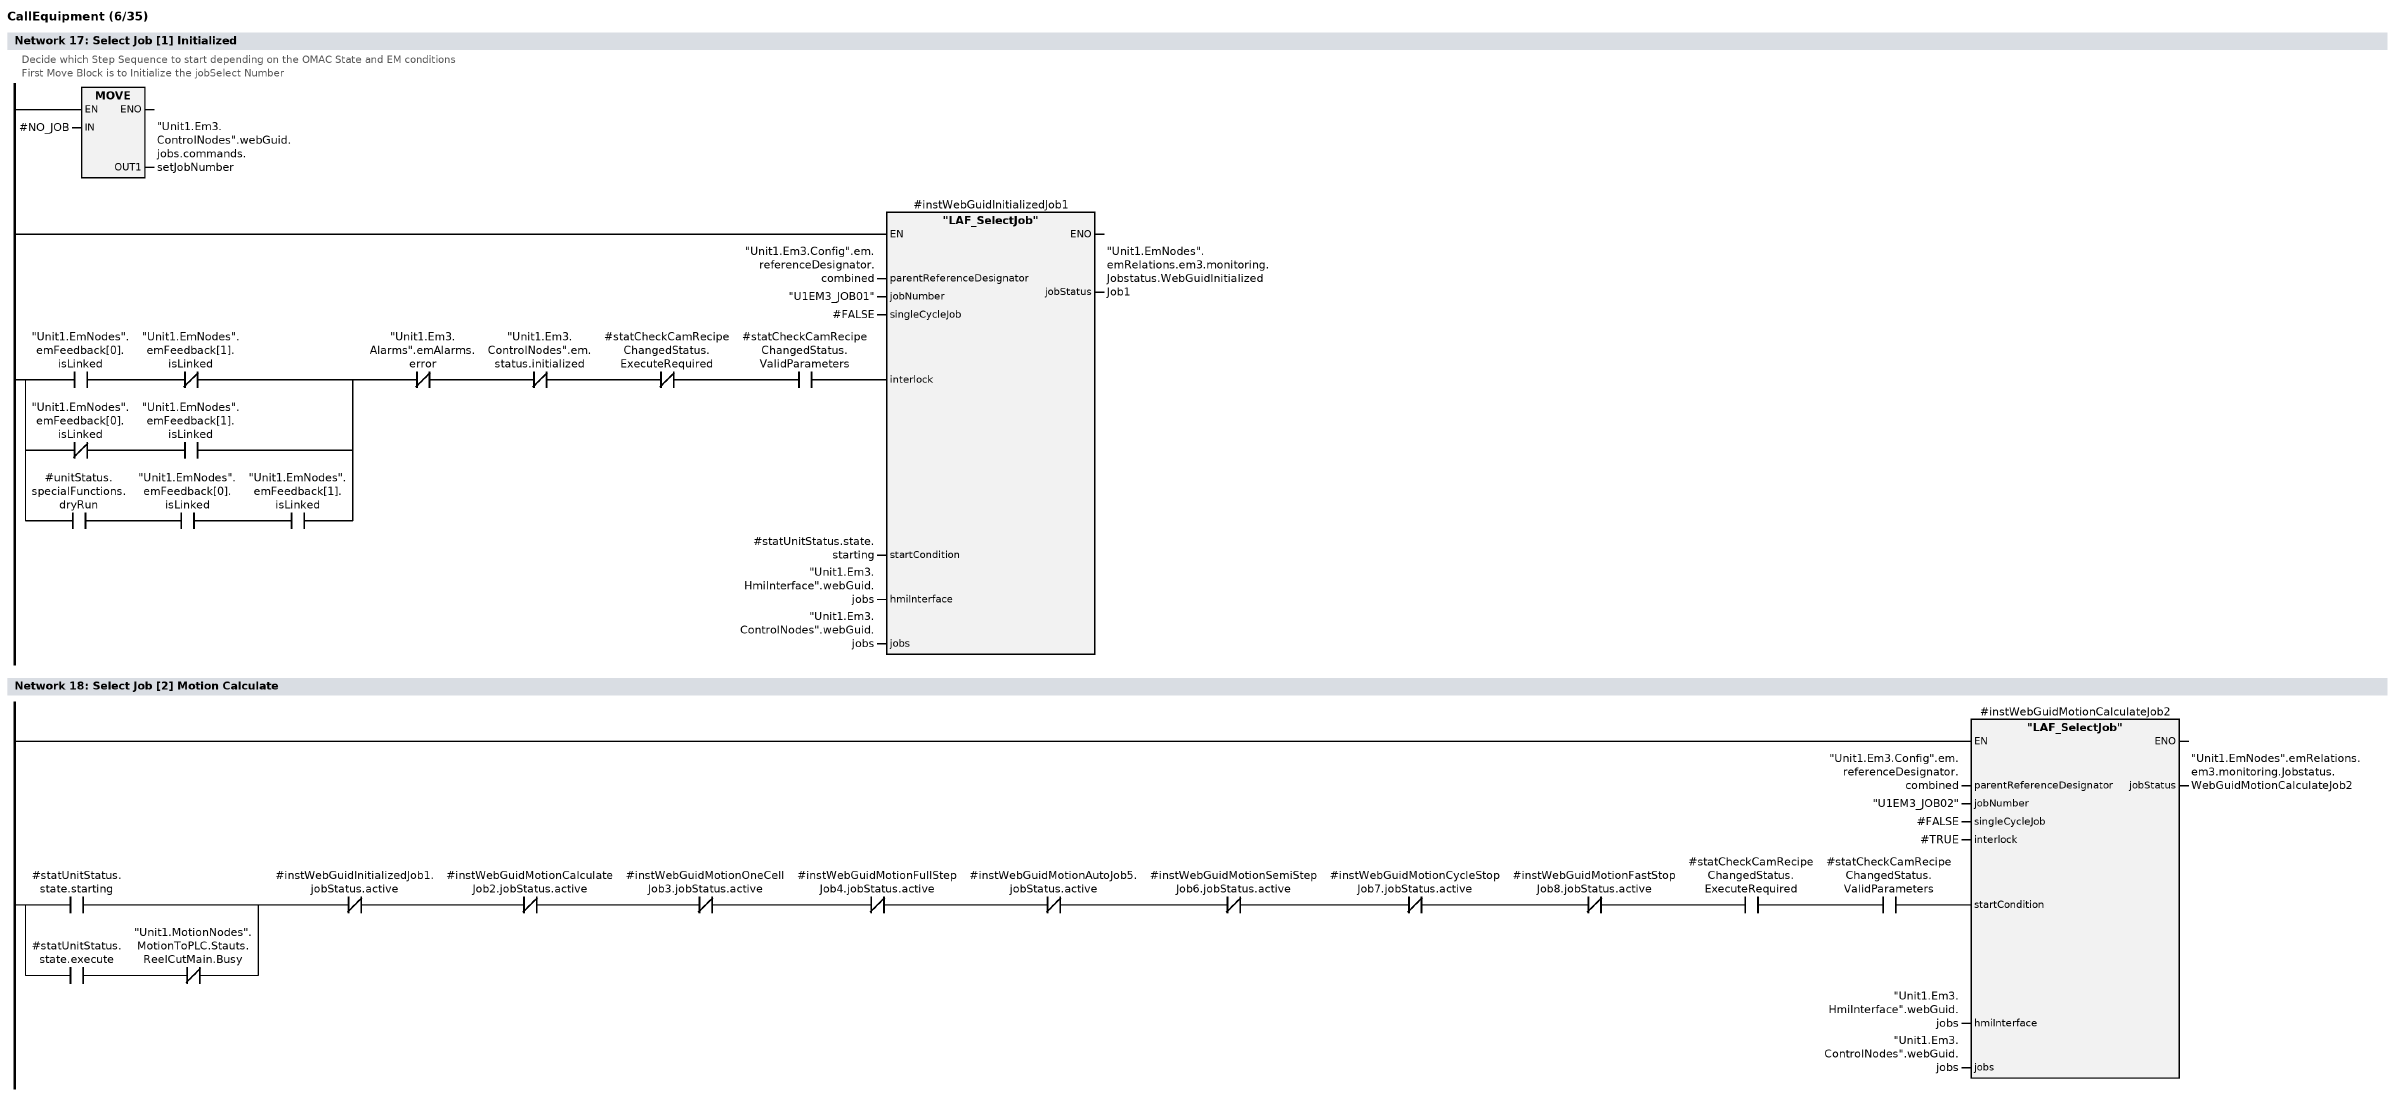
   RUNG wire#powerrail
      Move(in := #NO_JOB, out1 => "Unit1.Em3.ControlNodes".webGuid.jobs.commands.setJobNumber)
   END_RUNG
   RUNG wire#powerrail
      #instWebGuidInitializedJob1(interlock := wire#w2, parentReferenceDesignator := "Unit1.Em3.Config".em.referenceDesignator.combined, jobNumber := "U1EM3_JOB01", singleCycleJob := #FALSE, startCondition := #statUnitStatus.state.starting, hmiInterface := "Unit1.Em3.HmiInterface".webGuid.jobs, jobs := "Unit1.Em3.ControlNodes".webGuid.jobs, jobStatus => "Unit1.EmNodes".emRelations.em3.monitoring.Jobstatus.WebGuidInitializedJob1)
   END_RUNG
   RUNG wire#powerrail
      Contact( "Unit1.EmNodes".emFeedback[0].isLinked )
      I_Contact( "Unit1.EmNodes".emFeedback[1].isLinked )
      wire#w1
      I_Contact( "Unit1.Em3.Alarms".emAlarms.error )
      I_Contact( "Unit1.Em3.ControlNodes".em.status.initialized )
      I_Contact( #statCheckCamRecipeChangedStatus.ExecuteRequired )
      Contact( #statCheckCamRecipeChangedStatus.ValidParameters )
   END_RUNG wire#w2
   RUNG wire#powerrail
      I_Contact( "Unit1.EmNodes".emFeedback[0].isLinked )
      Contact( "Unit1.EmNodes".emFeedback[1].isLinked )
   END_RUNG wire#w1
   RUNG wire#powerrail
      Contact( #unitStatus.specialFunctions.dryRun )
      Contact( "Unit1.EmNodes".emFeedback[0].isLinked )
      Contact( "Unit1.EmNodes".emFeedback[1].isLinked )
   END_RUNG wire#w1
   // the same network as SCL:
   "Unit1.Em3.ControlNodes".webGuid.jobs.commands.setJobNumber := #NO_JOB;
   #instWebGuidInitializedJob1(parentReferenceDesignator := "Unit1.Em3.Config".em.referenceDesignator.combined,   // "LAF_SelectJob"
                           jobNumber := "U1EM3_JOB01",
                           singleCycleJob := #FALSE,
                           interlock := (("Unit1.EmNodes".emFeedback[0].isLinked AND NOT "Unit1.EmNodes".emFeedback[1].isLinked) OR (NOT "Unit1.EmNodes".emFeedback[0].isLinked AND "Unit1.EmNodes".emFeedback[1].isLinked) OR (#unitStatus.specialFunctions.dryRun AND "Unit1.EmNodes".emFeedback[0].isLinked AND "Unit1.EmNodes".emFeedback[1].isLinked)) AND NOT "Unit1.Em3.Alarms".emAlarms.error AND NOT "Unit1.Em3.ControlNodes".em.status.initialized AND NOT #statCheckCamRecipeChangedStatus.ExecuteRequired AND #statCheckCamRecipeChangedStatus.ValidParameters,
                           startCondition := #statUnitStatus.state.starting,
                           hmiInterface := "Unit1.Em3.HmiInterface".webGuid.jobs,
                           jobs := "Unit1.Em3.ControlNodes".webGuid.jobs,
                           jobStatus => "Unit1.EmNodes".emRelations.em3.monitoring.Jobstatus.WebGuidInitializedJob1);
END_REGION

REGION Network 18: Select Job [2] Motion Calculate
   RUNG wire#powerrail
      #instWebGuidMotionCalculateJob2(startCondition := wire#w2, parentReferenceDesignator := "Unit1.Em3.Config".em.referenceDesignator.combined, jobNumber := "U1EM3_JOB02", singleCycleJob := #FALSE, interlock := #TRUE, hmiInterface := "Unit1.Em3.HmiInterface".webGuid.jobs, jobs := "Unit1.Em3.ControlNodes".webGuid.jobs, jobStatus => "Unit1.EmNodes".emRelations.em3.monitoring.Jobstatus.WebGuidMotionCalculateJob2)
   END_RUNG
   RUNG wire#powerrail
      Contact( #statUnitStatus.state.starting )
      wire#w1
      I_Contact( #instWebGuidInitializedJob1.jobStatus.active )
      I_Contact( #instWebGuidMotionCalculateJob2.jobStatus.active )
      I_Contact( #instWebGuidMotionOneCellJob3.jobStatus.active )
      I_Contact( #instWebGuidMotionFullStepJob4.jobStatus.active )
      I_Contact( #instWebGuidMotionAutoJob5.jobStatus.active )
      I_Contact( #instWebGuidMotionSemiStepJob6.jobStatus.active )
      I_Contact( #instWebGuidMotionCycleStopJob7.jobStatus.active )
      I_Contact( #instWebGuidMotionFastStopJob8.jobStatus.active )
      Contact( #statCheckCamRecipeChangedStatus.ExecuteRequired )
      Contact( #statCheckCamRecipeChangedStatus.ValidParameters )
   END_RUNG wire#w2
   RUNG wire#powerrail
      Contact( #statUnitStatus.state.execute )
      I_Contact( "Unit1.MotionNodes".MotionToPLC.Stauts.ReelCutMain.Busy )
   END_RUNG wire#w1
   // the same network as SCL:
   #instWebGuidMotionCalculateJob2(parentReferenceDesignator := "Unit1.Em3.Config".em.referenceDesignator.combined,   // "LAF_SelectJob"
                           jobNumber := "U1EM3_JOB02",
                           singleCycleJob := #FALSE,
                           interlock := #TRUE,
                           startCondition := (#statUnitStatus.state.starting OR (#statUnitStatus.state.execute AND NOT "Unit1.MotionNodes".MotionToPLC.Stauts.ReelCutMain.Busy)) AND NOT #instWebGuidInitializedJob1.jobStatus.active AND NOT #instWebGuidMotionCalculateJob2.jobStatus.active AND NOT #instWebGuidMotionOneCellJob3.jobStatus.active AND NOT #instWebGuidMotionFullStepJob4.jobStatus.active AND NOT #instWebGuidMotionAutoJob5.jobStatus.active AND NOT #instWebGuidMotionSemiStepJob6.jobStatus.active AND NOT #instWebGuidMotionCycleStopJob7.jobStatus.active AND NOT #instWebGuidMotionFastStopJob8.jobStatus.active AND #statCheckCamRecipeChangedStatus.ExecuteRequired AND #statCheckCamRecipeChangedStatus.ValidParameters,
                           hmiInterface := "Unit1.Em3.HmiInterface".webGuid.jobs,
                           jobs := "Unit1.Em3.ControlNodes".webGuid.jobs,
                           jobStatus => "Unit1.EmNodes".emRelations.em3.monitoring.Jobstatus.WebGuidMotionCalculateJob2);
END_REGION

REGION Network 19: Select Job [3] Motion OneCell
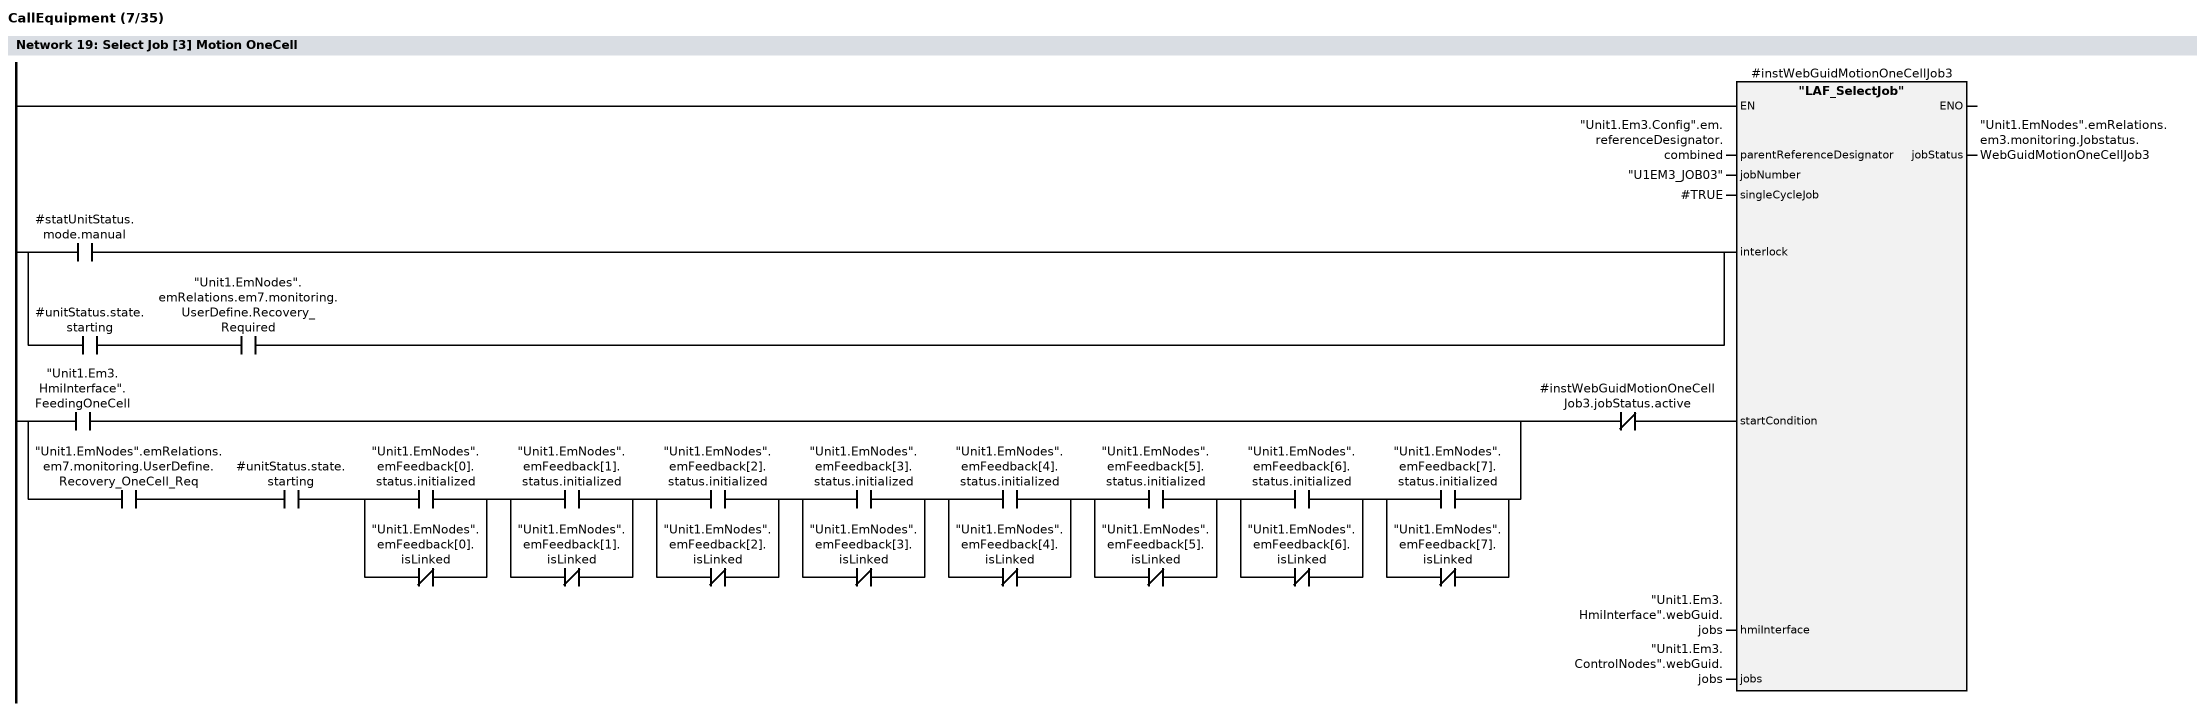
   RUNG wire#powerrail
      #instWebGuidMotionOneCellJob3(interlock := wire#w1, startCondition := wire#w11, parentReferenceDesignator := "Unit1.Em3.Config".em.referenceDesignator.combined, jobNumber := "U1EM3_JOB03", singleCycleJob := #TRUE, hmiInterface := "Unit1.Em3.HmiInterface".webGuid.jobs, jobs := "Unit1.Em3.ControlNodes".webGuid.jobs, jobStatus => "Unit1.EmNodes".emRelations.em3.monitoring.Jobstatus.WebGuidMotionOneCellJob3)
   END_RUNG
   RUNG wire#powerrail
      Contact( #statUnitStatus.mode.manual )
   END_RUNG wire#w1
   RUNG wire#powerrail
      Contact( #unitStatus.state.starting )
      Contact( "Unit1.EmNodes".emRelations.em7.monitoring.UserDefine.Recovery_Required )
   END_RUNG wire#w1
   RUNG wire#powerrail
      Contact( "Unit1.Em3.HmiInterface".FeedingOneCell )
      wire#w2
      I_Contact( #instWebGuidMotionOneCellJob3.jobStatus.active )
   END_RUNG wire#w11
   RUNG wire#powerrail
      Contact( "Unit1.EmNodes".emRelations.em7.monitoring.UserDefine.Recovery_OneCell_Req )
      Contact( #unitStatus.state.starting )
      wire#w3
      Contact( "Unit1.EmNodes".emFeedback[0].status.initialized )
      wire#w4
      Contact( "Unit1.EmNodes".emFeedback[1].status.initialized )
      wire#w5
      Contact( "Unit1.EmNodes".emFeedback[2].status.initialized )
      wire#w6
      Contact( "Unit1.EmNodes".emFeedback[3].status.initialized )
      wire#w7
      Contact( "Unit1.EmNodes".emFeedback[4].status.initialized )
      wire#w8
      Contact( "Unit1.EmNodes".emFeedback[5].status.initialized )
      wire#w9
      Contact( "Unit1.EmNodes".emFeedback[6].status.initialized )
      wire#w10
      Contact( "Unit1.EmNodes".emFeedback[7].status.initialized )
   END_RUNG wire#w2
   RUNG wire#w3
      I_Contact( "Unit1.EmNodes".emFeedback[0].isLinked )
   END_RUNG wire#w4
   RUNG wire#w4
      I_Contact( "Unit1.EmNodes".emFeedback[1].isLinked )
   END_RUNG wire#w5
   RUNG wire#w5
      I_Contact( "Unit1.EmNodes".emFeedback[2].isLinked )
   END_RUNG wire#w6
   RUNG wire#w6
      I_Contact( "Unit1.EmNodes".emFeedback[3].isLinked )
   END_RUNG wire#w7
   RUNG wire#w7
      I_Contact( "Unit1.EmNodes".emFeedback[4].isLinked )
   END_RUNG wire#w8
   RUNG wire#w8
      I_Contact( "Unit1.EmNodes".emFeedback[5].isLinked )
   END_RUNG wire#w9
   RUNG wire#w9
      I_Contact( "Unit1.EmNodes".emFeedback[6].isLinked )
   END_RUNG wire#w10
   RUNG wire#w10
      I_Contact( "Unit1.EmNodes".emFeedback[7].isLinked )
   END_RUNG wire#w2
   // the same network as SCL:
   #instWebGuidMotionOneCellJob3(parentReferenceDesignator := "Unit1.Em3.Config".em.referenceDesignator.combined,   // "LAF_SelectJob"
                           jobNumber := "U1EM3_JOB03",
                           singleCycleJob := #TRUE,
                           interlock := #statUnitStatus.mode.manual OR (#unitStatus.state.starting AND "Unit1.EmNodes".emRelations.em7.monitoring.UserDefine.Recovery_Required),
                           startCondition := ("Unit1.Em3.HmiInterface".FeedingOneCell OR ("Unit1.EmNodes".emRelations.em7.monitoring.UserDefine.Recovery_OneCell_Req AND #unitStatus.state.starting AND ("Unit1.EmNodes".emFeedback[0].status.initialized OR NOT "Unit1.EmNodes".emFeedback[0].isLinked) AND ("Unit1.EmNodes".emFeedback[1].status.initialized OR NOT "Unit1.EmNodes".emFeedback[1].isLinked) AND ("Unit1.EmNodes".emFeedback[2].status.initialized OR NOT "Unit1.EmNodes".emFeedback[2].isLinked) AND ("Unit1.EmNodes".emFeedback[3].status.initialized OR NOT "Unit1.EmNodes".emFeedback[3].isLinked) AND ("Unit1.EmNodes".emFeedback[4].status.initialized OR NOT "Unit1.EmNodes".emFeedback[4].isLinked) AND ("Unit1.EmNodes".emFeedback[5].status.initialized OR NOT "Unit1.EmNodes".emFeedback[5].isLinked) AND ("Unit1.EmNodes".emFeedback[6].status.initialized OR NOT "Unit1.EmNodes".emFeedback[6].isLinked) AND ("Unit1.EmNodes".emFeedback[7].status.initialized OR NOT "Unit1.EmNodes".emFeedback[7].isLinked))) AND NOT #instWebGuidMotionOneCellJob3.jobStatus.active,
                           hmiInterface := "Unit1.Em3.HmiInterface".webGuid.jobs,
                           jobs := "Unit1.Em3.ControlNodes".webGuid.jobs,
                           jobStatus => "Unit1.EmNodes".emRelations.em3.monitoring.Jobstatus.WebGuidMotionOneCellJob3);
END_REGION

REGION Network 20: Select Job [4] Motion FullStep
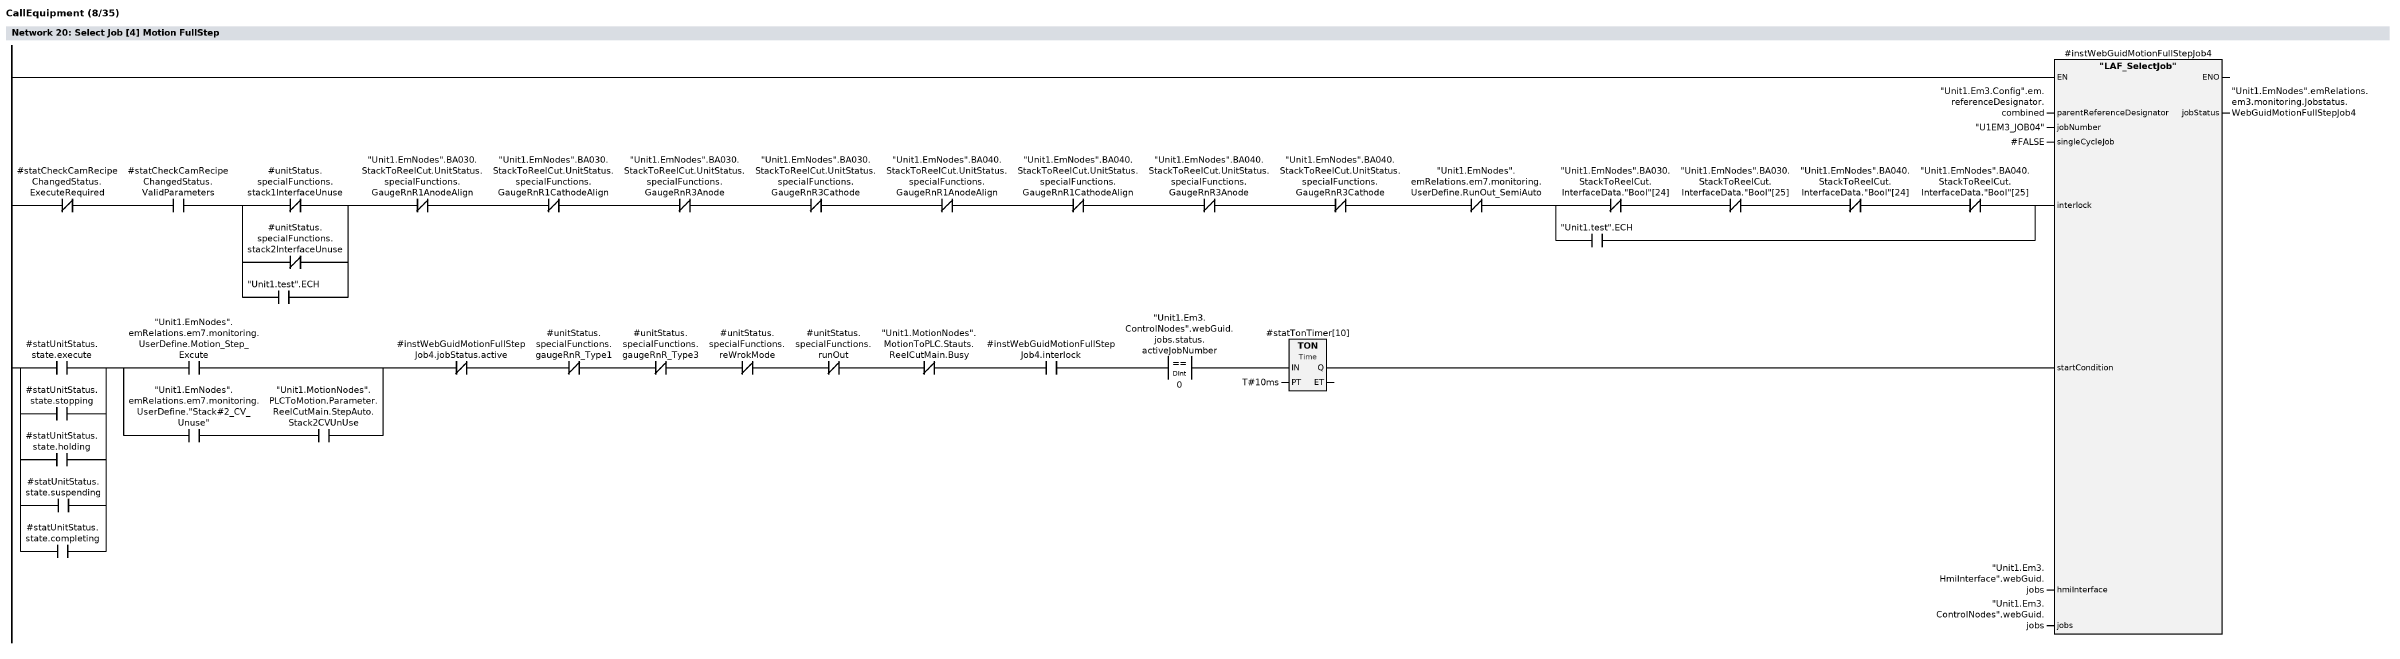
   RUNG wire#powerrail
      #instWebGuidMotionFullStepJob4(interlock := wire#w4, startCondition := wire#w7, parentReferenceDesignator := "Unit1.Em3.Config".em.referenceDesignator.combined, jobNumber := "U1EM3_JOB04", singleCycleJob := #FALSE, hmiInterface := "Unit1.Em3.HmiInterface".webGuid.jobs, jobs := "Unit1.Em3.ControlNodes".webGuid.jobs, jobStatus => "Unit1.EmNodes".emRelations.em3.monitoring.Jobstatus.WebGuidMotionFullStepJob4)
   END_RUNG
   RUNG wire#powerrail
      I_Contact( #statCheckCamRecipeChangedStatus.ExecuteRequired )
      Contact( #statCheckCamRecipeChangedStatus.ValidParameters )
      wire#w1
      I_Contact( #unitStatus.specialFunctions.stack1InterfaceUnuse )
      wire#w2
      I_Contact( "Unit1.EmNodes".BA030.StackToReelCut.UnitStatus.specialFunctions.GaugeRnR1AnodeAlign )
      I_Contact( "Unit1.EmNodes".BA030.StackToReelCut.UnitStatus.specialFunctions.GaugeRnR1CathodeAlign )
      I_Contact( "Unit1.EmNodes".BA030.StackToReelCut.UnitStatus.specialFunctions.GaugeRnR3Anode )
      I_Contact( "Unit1.EmNodes".BA030.StackToReelCut.UnitStatus.specialFunctions.GaugeRnR3Cathode )
      I_Contact( "Unit1.EmNodes".BA040.StackToReelCut.UnitStatus.specialFunctions.GaugeRnR1AnodeAlign )
      I_Contact( "Unit1.EmNodes".BA040.StackToReelCut.UnitStatus.specialFunctions.GaugeRnR1CathodeAlign )
      I_Contact( "Unit1.EmNodes".BA040.StackToReelCut.UnitStatus.specialFunctions.GaugeRnR3Anode )
      I_Contact( "Unit1.EmNodes".BA040.StackToReelCut.UnitStatus.specialFunctions.GaugeRnR3Cathode )
      I_Contact( "Unit1.EmNodes".emRelations.em7.monitoring.UserDefine.RunOut_SemiAuto )
      wire#w3
      I_Contact( "Unit1.EmNodes".BA030.StackToReelCut.InterfaceData."Bool"[24] )
      I_Contact( "Unit1.EmNodes".BA030.StackToReelCut.InterfaceData."Bool"[25] )
      I_Contact( "Unit1.EmNodes".BA040.StackToReelCut.InterfaceData."Bool"[24] )
      I_Contact( "Unit1.EmNodes".BA040.StackToReelCut.InterfaceData."Bool"[25] )
   END_RUNG wire#w4
   RUNG wire#w1
      I_Contact( #unitStatus.specialFunctions.stack2InterfaceUnuse )
   END_RUNG wire#w2
   RUNG wire#w1
      Contact( "Unit1.test".ECH )
   END_RUNG wire#w2
   RUNG wire#w3
      Contact( "Unit1.test".ECH )
   END_RUNG wire#w4
   RUNG wire#powerrail
      Contact( #statUnitStatus.state.execute )
      wire#w5
      Contact( "Unit1.EmNodes".emRelations.em7.monitoring.UserDefine.Motion_Step_Excute )
      wire#w6
      I_Contact( #instWebGuidMotionFullStepJob4.jobStatus.active )
      I_Contact( #unitStatus.specialFunctions.gaugeRnR_Type1 )
      I_Contact( #unitStatus.specialFunctions.gaugeRnR_Type3 )
      I_Contact( #unitStatus.specialFunctions.reWrokMode )
      I_Contact( #unitStatus.specialFunctions.runOut )
      I_Contact( "Unit1.MotionNodes".MotionToPLC.Stauts.ReelCutMain.Busy )
      Contact( #instWebGuidMotionFullStepJob4.interlock )
      { S7_Templates := "SrcType := DInt" } EQ_Contact(in1 := "Unit1.Em3.ControlNodes".webGuid.jobs.status.activeJobNumber, in2 := 0)
      { S7_Templates := "time_type := Time" } #statTonTimer[10].TON(pt := T#10ms, et =>)
   END_RUNG wire#w7
   RUNG wire#powerrail
      Contact( #statUnitStatus.state.stopping )
   END_RUNG wire#w5
   RUNG wire#powerrail
      Contact( #statUnitStatus.state.holding )
   END_RUNG wire#w5
   RUNG wire#powerrail
      Contact( #statUnitStatus.state.suspending )
   END_RUNG wire#w5
   RUNG wire#powerrail
      Contact( #statUnitStatus.state.completing )
   END_RUNG wire#w5
   RUNG wire#w5
      Contact( "Unit1.EmNodes".emRelations.em7.monitoring.UserDefine."Stack#2_CV_Unuse" )
      Contact( "Unit1.MotionNodes".PLCToMotion.Parameter.ReelCutMain.StepAuto.Stack2CVUnUse )
   END_RUNG wire#w6
   // the same network as SCL:
   #statTonTimer[10].TON(IN := (#statUnitStatus.state.execute OR #statUnitStatus.state.stopping OR #statUnitStatus.state.holding OR #statUnitStatus.state.suspending OR #statUnitStatus.state.completing) AND ("Unit1.EmNodes".emRelations.em7.monitoring.UserDefine.Motion_Step_Excute OR ("Unit1.EmNodes".emRelations.em7.monitoring.UserDefine."Stack#2_CV_Unuse" AND "Unit1.MotionNodes".PLCToMotion.Parameter.ReelCutMain.StepAuto.Stack2CVUnUse)) AND NOT #instWebGuidMotionFullStepJob4.jobStatus.active AND NOT #unitStatus.specialFunctions.gaugeRnR_Type1 AND NOT #unitStatus.specialFunctions.gaugeRnR_Type3 AND NOT #unitStatus.specialFunctions.reWrokMode AND NOT #unitStatus.specialFunctions.runOut AND NOT "Unit1.MotionNodes".MotionToPLC.Stauts.ReelCutMain.Busy AND #instWebGuidMotionFullStepJob4.interlock AND ("Unit1.Em3.ControlNodes".webGuid.jobs.status.activeJobNumber = 0),
                         PT := T#10ms);
   #instWebGuidMotionFullStepJob4(parentReferenceDesignator := "Unit1.Em3.Config".em.referenceDesignator.combined,   // "LAF_SelectJob"
                           jobNumber := "U1EM3_JOB04",
                           singleCycleJob := #FALSE,
                           interlock := NOT #statCheckCamRecipeChangedStatus.ExecuteRequired AND #statCheckCamRecipeChangedStatus.ValidParameters AND (NOT #unitStatus.specialFunctions.stack1InterfaceUnuse OR NOT #unitStatus.specialFunctions.stack2InterfaceUnuse OR "Unit1.test".ECH) AND NOT "Unit1.EmNodes".BA030.StackToReelCut.UnitStatus.specialFunctions.GaugeRnR1AnodeAlign AND NOT "Unit1.EmNodes".BA030.StackToReelCut.UnitStatus.specialFunctions.GaugeRnR1CathodeAlign AND NOT "Unit1.EmNodes".BA030.StackToReelCut.UnitStatus.specialFunctions.GaugeRnR3Anode AND NOT "Unit1.EmNodes".BA030.StackToReelCut.UnitStatus.specialFunctions.GaugeRnR3Cathode AND NOT "Unit1.EmNodes".BA040.StackToReelCut.UnitStatus.specialFunctions.GaugeRnR1AnodeAlign AND NOT "Unit1.EmNodes".BA040.StackToReelCut.UnitStatus.specialFunctions.GaugeRnR1CathodeAlign AND NOT "Unit1.EmNodes".BA040.StackToReelCut.UnitStatus.specialFunctions.GaugeRnR3Anode AND NOT "Unit1.EmNodes".BA040.StackToReelCut.UnitStatus.specialFunctions.GaugeRnR3Cathode AND NOT "Unit1.EmNodes".emRelations.em7.monitoring.UserDefine.RunOut_SemiAuto AND ((NOT "Unit1.EmNodes".BA030.StackToReelCut.InterfaceData."Bool"[24] AND NOT "Unit1.EmNodes".BA030.StackToReelCut.InterfaceData."Bool"[25] AND NOT "Unit1.EmNodes".BA040.StackToReelCut.InterfaceData."Bool"[24] AND NOT "Unit1.EmNodes".BA040.StackToReelCut.InterfaceData."Bool"[25]) OR "Unit1.test".ECH),
                           startCondition := #statTonTimer[10].Q,
                           hmiInterface := "Unit1.Em3.HmiInterface".webGuid.jobs,
                           jobs := "Unit1.Em3.ControlNodes".webGuid.jobs,
                           jobStatus => "Unit1.EmNodes".emRelations.em3.monitoring.Jobstatus.WebGuidMotionFullStepJob4);
END_REGION

REGION Network 21: Select Job [5] Motion Auto
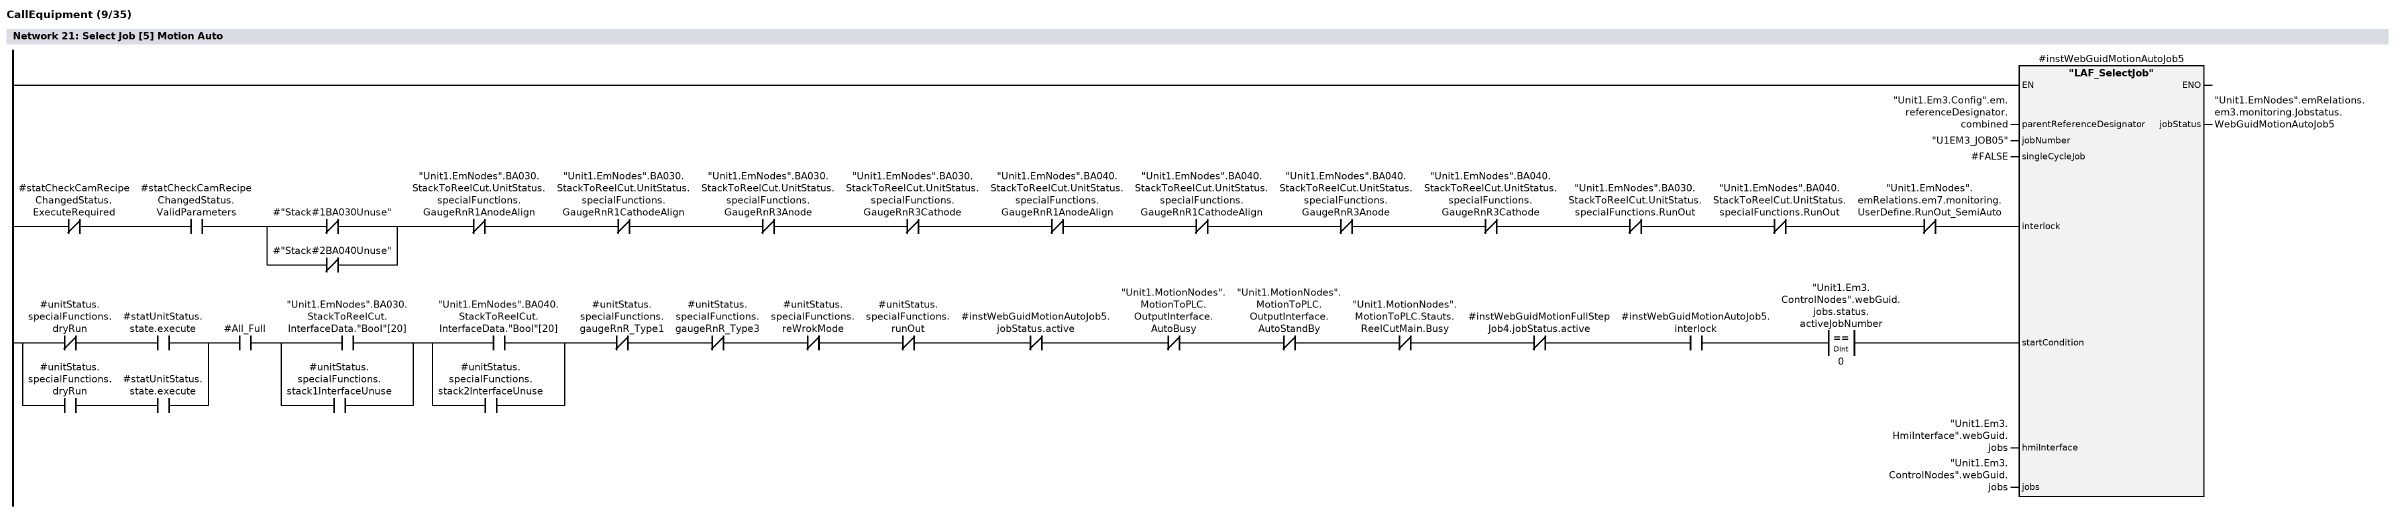
   RUNG wire#powerrail
      #instWebGuidMotionAutoJob5(interlock := wire#w3, startCondition := wire#w8, parentReferenceDesignator := "Unit1.Em3.Config".em.referenceDesignator.combined, jobNumber := "U1EM3_JOB05", singleCycleJob := #FALSE, hmiInterface := "Unit1.Em3.HmiInterface".webGuid.jobs, jobs := "Unit1.Em3.ControlNodes".webGuid.jobs, jobStatus => "Unit1.EmNodes".emRelations.em3.monitoring.Jobstatus.WebGuidMotionAutoJob5)
   END_RUNG
   RUNG wire#powerrail
      I_Contact( #statCheckCamRecipeChangedStatus.ExecuteRequired )
      Contact( #statCheckCamRecipeChangedStatus.ValidParameters )
      wire#w1
      I_Contact( #"Stack#1BA030Unuse" )
      wire#w2
      I_Contact( "Unit1.EmNodes".BA030.StackToReelCut.UnitStatus.specialFunctions.GaugeRnR1AnodeAlign )
      I_Contact( "Unit1.EmNodes".BA030.StackToReelCut.UnitStatus.specialFunctions.GaugeRnR1CathodeAlign )
      I_Contact( "Unit1.EmNodes".BA030.StackToReelCut.UnitStatus.specialFunctions.GaugeRnR3Anode )
      I_Contact( "Unit1.EmNodes".BA030.StackToReelCut.UnitStatus.specialFunctions.GaugeRnR3Cathode )
      I_Contact( "Unit1.EmNodes".BA040.StackToReelCut.UnitStatus.specialFunctions.GaugeRnR1AnodeAlign )
      I_Contact( "Unit1.EmNodes".BA040.StackToReelCut.UnitStatus.specialFunctions.GaugeRnR1CathodeAlign )
      I_Contact( "Unit1.EmNodes".BA040.StackToReelCut.UnitStatus.specialFunctions.GaugeRnR3Anode )
      I_Contact( "Unit1.EmNodes".BA040.StackToReelCut.UnitStatus.specialFunctions.GaugeRnR3Cathode )
      I_Contact( "Unit1.EmNodes".BA030.StackToReelCut.UnitStatus.specialFunctions.RunOut )
      I_Contact( "Unit1.EmNodes".BA040.StackToReelCut.UnitStatus.specialFunctions.RunOut )
      I_Contact( "Unit1.EmNodes".emRelations.em7.monitoring.UserDefine.RunOut_SemiAuto )
   END_RUNG wire#w3
   RUNG wire#w1
      I_Contact( #"Stack#2BA040Unuse" )
   END_RUNG wire#w2
   RUNG wire#powerrail
      I_Contact( #unitStatus.specialFunctions.dryRun )
      Contact( #statUnitStatus.state.execute )
      wire#w4
      Contact( #All_Full )
      wire#w5
      Contact( "Unit1.EmNodes".BA030.StackToReelCut.InterfaceData."Bool"[20] )
      wire#w6
      Contact( "Unit1.EmNodes".BA040.StackToReelCut.InterfaceData."Bool"[20] )
      wire#w7
      I_Contact( #unitStatus.specialFunctions.gaugeRnR_Type1 )
      I_Contact( #unitStatus.specialFunctions.gaugeRnR_Type3 )
      I_Contact( #unitStatus.specialFunctions.reWrokMode )
      I_Contact( #unitStatus.specialFunctions.runOut )
      I_Contact( #instWebGuidMotionAutoJob5.jobStatus.active )
      I_Contact( "Unit1.MotionNodes".MotionToPLC.OutputInterface.AutoBusy )
      I_Contact( "Unit1.MotionNodes".MotionToPLC.OutputInterface.AutoStandBy )
      I_Contact( "Unit1.MotionNodes".MotionToPLC.Stauts.ReelCutMain.Busy )
      I_Contact( #instWebGuidMotionFullStepJob4.jobStatus.active )
      Contact( #instWebGuidMotionAutoJob5.interlock )
      { S7_Templates := "SrcType := DInt" } EQ_Contact(in1 := "Unit1.Em3.ControlNodes".webGuid.jobs.status.activeJobNumber, in2 := 0)
   END_RUNG wire#w8
   RUNG wire#powerrail
      Contact( #unitStatus.specialFunctions.dryRun )
      Contact( #statUnitStatus.state.execute )
   END_RUNG wire#w4
   RUNG wire#w5
      Contact( #unitStatus.specialFunctions.stack1InterfaceUnuse )
   END_RUNG wire#w6
   RUNG wire#w6
      Contact( #unitStatus.specialFunctions.stack2InterfaceUnuse )
   END_RUNG wire#w7
   // the same network as SCL:
   #instWebGuidMotionAutoJob5(parentReferenceDesignator := "Unit1.Em3.Config".em.referenceDesignator.combined,   // "LAF_SelectJob"
                           jobNumber := "U1EM3_JOB05",
                           singleCycleJob := #FALSE,
                           interlock := NOT #statCheckCamRecipeChangedStatus.ExecuteRequired AND #statCheckCamRecipeChangedStatus.ValidParameters AND (NOT #"Stack#1BA030Unuse" OR NOT #"Stack#2BA040Unuse") AND NOT "Unit1.EmNodes".BA030.StackToReelCut.UnitStatus.specialFunctions.GaugeRnR1AnodeAlign AND NOT "Unit1.EmNodes".BA030.StackToReelCut.UnitStatus.specialFunctions.GaugeRnR1CathodeAlign AND NOT "Unit1.EmNodes".BA030.StackToReelCut.UnitStatus.specialFunctions.GaugeRnR3Anode AND NOT "Unit1.EmNodes".BA030.StackToReelCut.UnitStatus.specialFunctions.GaugeRnR3Cathode AND NOT "Unit1.EmNodes".BA040.StackToReelCut.UnitStatus.specialFunctions.GaugeRnR1AnodeAlign AND NOT "Unit1.EmNodes".BA040.StackToReelCut.UnitStatus.specialFunctions.GaugeRnR1CathodeAlign AND NOT "Unit1.EmNodes".BA040.StackToReelCut.UnitStatus.specialFunctions.GaugeRnR3Anode AND NOT "Unit1.EmNodes".BA040.StackToReelCut.UnitStatus.specialFunctions.GaugeRnR3Cathode AND NOT "Unit1.EmNodes".BA030.StackToReelCut.UnitStatus.specialFunctions.RunOut AND NOT "Unit1.EmNodes".BA040.StackToReelCut.UnitStatus.specialFunctions.RunOut AND NOT "Unit1.EmNodes".emRelations.em7.monitoring.UserDefine.RunOut_SemiAuto,
                           startCondition := ((NOT #unitStatus.specialFunctions.dryRun AND #statUnitStatus.state.execute) OR (#unitStatus.specialFunctions.dryRun AND #statUnitStatus.state.execute)) AND #All_Full AND ("Unit1.EmNodes".BA030.StackToReelCut.InterfaceData."Bool"[20] OR #unitStatus.specialFunctions.stack1InterfaceUnuse) AND ("Unit1.EmNodes".BA040.StackToReelCut.InterfaceData."Bool"[20] OR #unitStatus.specialFunctions.stack2InterfaceUnuse) AND NOT #unitStatus.specialFunctions.gaugeRnR_Type1 AND NOT #unitStatus.specialFunctions.gaugeRnR_Type3 AND NOT #unitStatus.specialFunctions.reWrokMode AND NOT #unitStatus.specialFunctions.runOut AND NOT #instWebGuidMotionAutoJob5.jobStatus.active AND NOT "Unit1.MotionNodes".MotionToPLC.OutputInterface.AutoBusy AND NOT "Unit1.MotionNodes".MotionToPLC.OutputInterface.AutoStandBy AND NOT "Unit1.MotionNodes".MotionToPLC.Stauts.ReelCutMain.Busy AND NOT #instWebGuidMotionFullStepJob4.jobStatus.active AND #instWebGuidMotionAutoJob5.interlock AND ("Unit1.Em3.ControlNodes".webGuid.jobs.status.activeJobNumber = 0),
                           hmiInterface := "Unit1.Em3.HmiInterface".webGuid.jobs,
                           jobs := "Unit1.Em3.ControlNodes".webGuid.jobs,
                           jobStatus => "Unit1.EmNodes".emRelations.em3.monitoring.Jobstatus.WebGuidMotionAutoJob5);
END_REGION

REGION Network 22: Select Job [6] Motion SemiStep
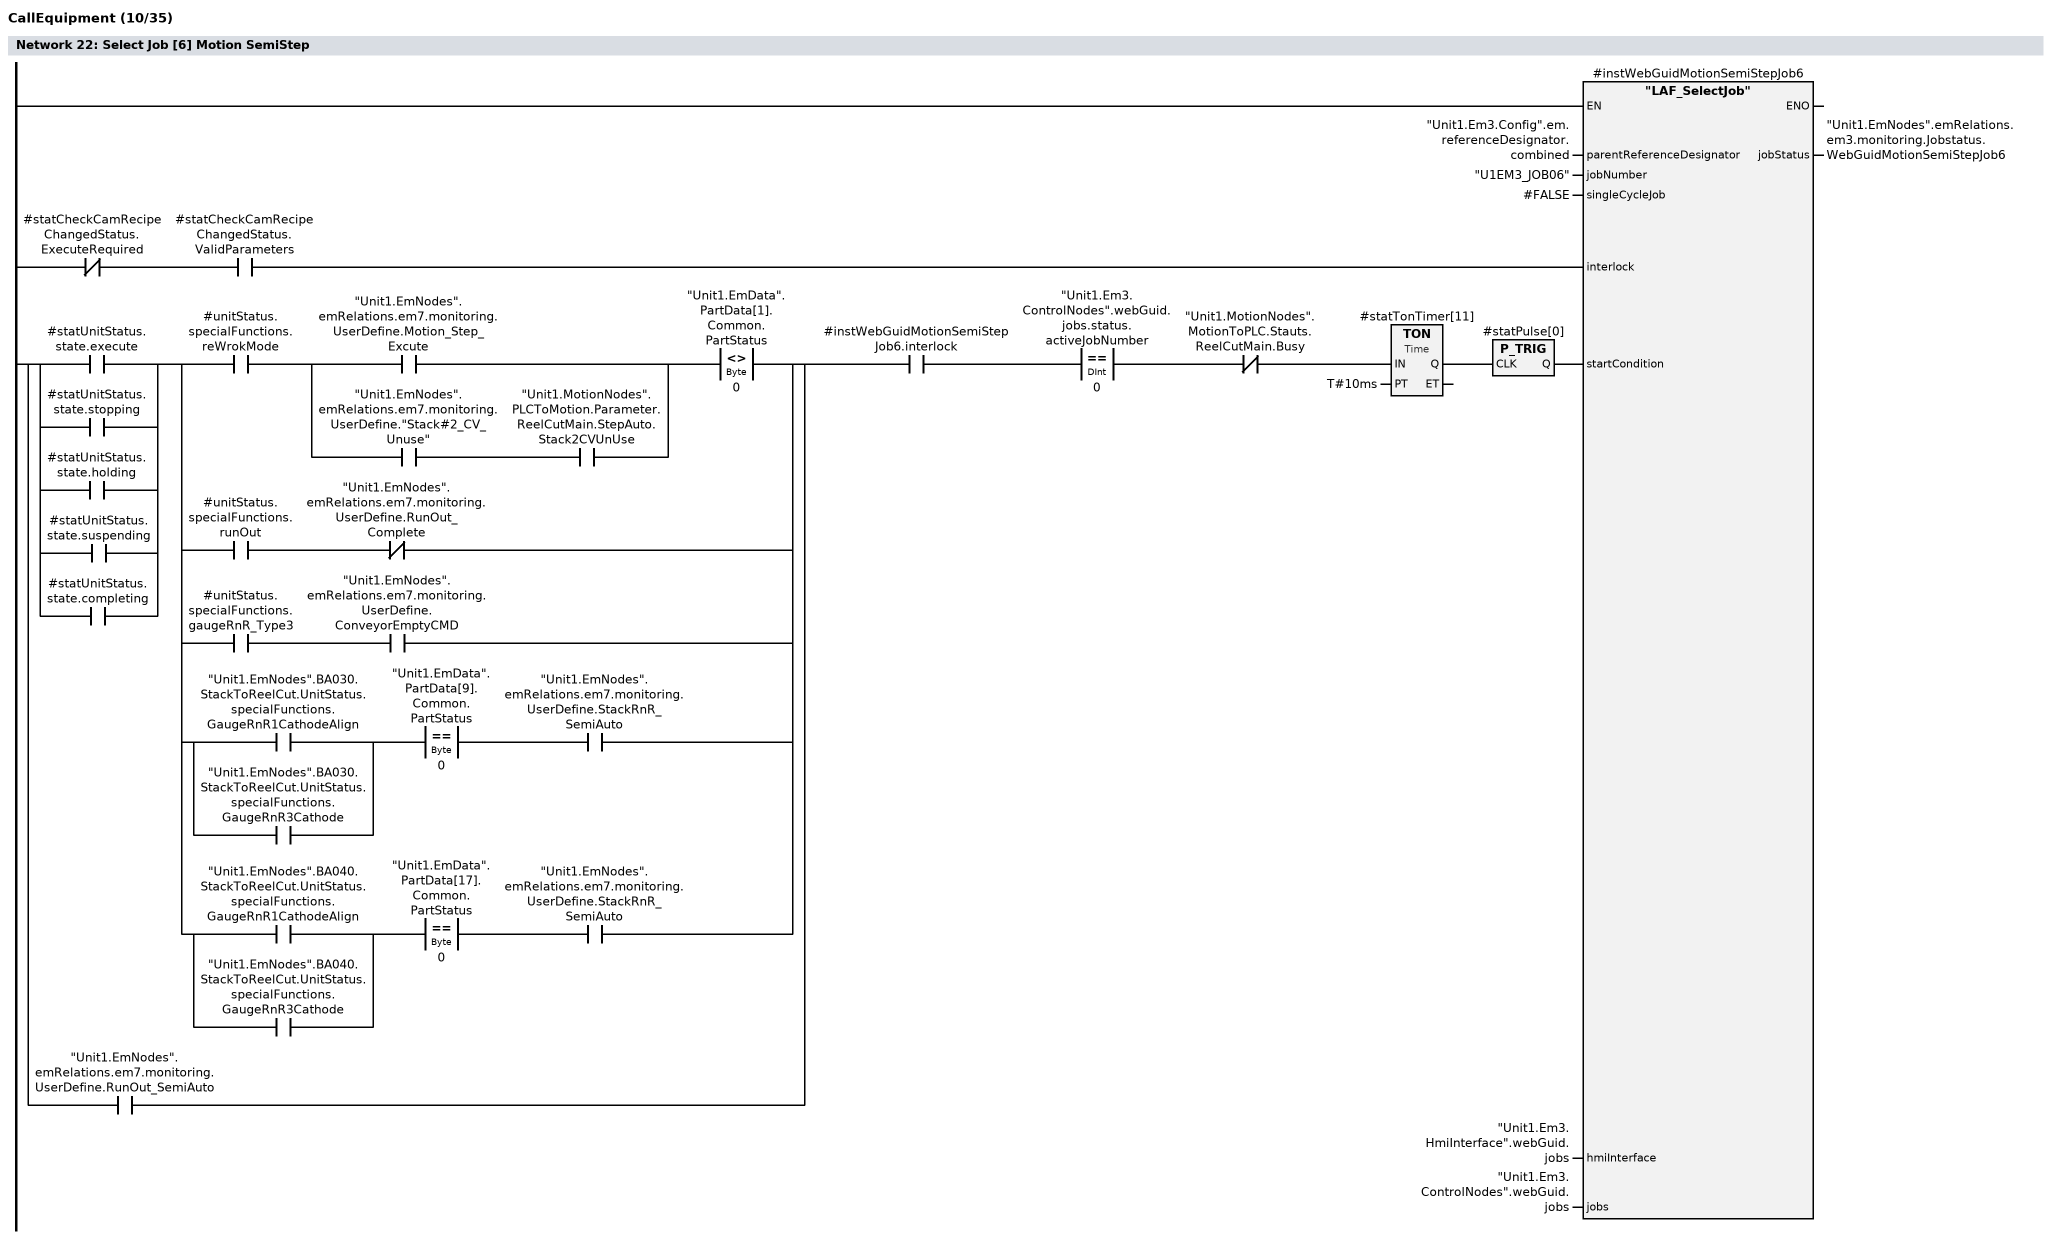
   RUNG wire#powerrail
      #instWebGuidMotionSemiStepJob6(interlock := wire#w1, startCondition := wire#w8, parentReferenceDesignator := "Unit1.Em3.Config".em.referenceDesignator.combined, jobNumber := "U1EM3_JOB06", singleCycleJob := #FALSE, hmiInterface := "Unit1.Em3.HmiInterface".webGuid.jobs, jobs := "Unit1.Em3.ControlNodes".webGuid.jobs, jobStatus => "Unit1.EmNodes".emRelations.em3.monitoring.Jobstatus.WebGuidMotionSemiStepJob6)
   END_RUNG
   RUNG wire#powerrail
      I_Contact( #statCheckCamRecipeChangedStatus.ExecuteRequired )
      Contact( #statCheckCamRecipeChangedStatus.ValidParameters )
   END_RUNG wire#w1
   RUNG wire#powerrail
      Contact( #statUnitStatus.state.execute )
      wire#w2
      Contact( #unitStatus.specialFunctions.reWrokMode )
      wire#w3
      Contact( "Unit1.EmNodes".emRelations.em7.monitoring.UserDefine.Motion_Step_Excute )
      wire#w4
      { S7_Templates := "SrcType := Byte" } NE_Contact(in1 := "Unit1.EmData".PartData[1].Common.PartStatus, in2 := 0)
      wire#w5
      Contact( #instWebGuidMotionSemiStepJob6.interlock )
      { S7_Templates := "SrcType := DInt" } EQ_Contact(in1 := "Unit1.Em3.ControlNodes".webGuid.jobs.status.activeJobNumber, in2 := 0)
      I_Contact( "Unit1.MotionNodes".MotionToPLC.Stauts.ReelCutMain.Busy )
      { S7_Templates := "time_type := Time" } #statTonTimer[11].TON(pt := T#10ms, et =>)
      P_Trig( #statPulse[0] )
   END_RUNG wire#w8
   RUNG wire#powerrail
      Contact( #statUnitStatus.state.stopping )
   END_RUNG wire#w2
   RUNG wire#powerrail
      Contact( #statUnitStatus.state.holding )
   END_RUNG wire#w2
   RUNG wire#powerrail
      Contact( #statUnitStatus.state.suspending )
   END_RUNG wire#w2
   RUNG wire#powerrail
      Contact( #statUnitStatus.state.completing )
   END_RUNG wire#w2
   RUNG wire#w3
      Contact( "Unit1.EmNodes".emRelations.em7.monitoring.UserDefine."Stack#2_CV_Unuse" )
      Contact( "Unit1.MotionNodes".PLCToMotion.Parameter.ReelCutMain.StepAuto.Stack2CVUnUse )
   END_RUNG wire#w4
   RUNG wire#w2
      Contact( #unitStatus.specialFunctions.runOut )
      I_Contact( "Unit1.EmNodes".emRelations.em7.monitoring.UserDefine.RunOut_Complete )
   END_RUNG wire#w5
   RUNG wire#w2
      Contact( #unitStatus.specialFunctions.gaugeRnR_Type3 )
      Contact( "Unit1.EmNodes".emRelations.em7.monitoring.UserDefine.ConveyorEmptyCMD )
   END_RUNG wire#w5
   RUNG wire#w2
      Contact( "Unit1.EmNodes".BA030.StackToReelCut.UnitStatus.specialFunctions.GaugeRnR1CathodeAlign )
      wire#w6
      { S7_Templates := "SrcType := Byte" } EQ_Contact(in1 := "Unit1.EmData".PartData[9].Common.PartStatus, in2 := 0)
      Contact( "Unit1.EmNodes".emRelations.em7.monitoring.UserDefine.StackRnR_SemiAuto )
   END_RUNG wire#w5
   RUNG wire#w2
      Contact( "Unit1.EmNodes".BA030.StackToReelCut.UnitStatus.specialFunctions.GaugeRnR3Cathode )
   END_RUNG wire#w6
   RUNG wire#w2
      Contact( "Unit1.EmNodes".BA040.StackToReelCut.UnitStatus.specialFunctions.GaugeRnR1CathodeAlign )
      wire#w7
      { S7_Templates := "SrcType := Byte" } EQ_Contact(in1 := "Unit1.EmData".PartData[17].Common.PartStatus, in2 := 0)
      Contact( "Unit1.EmNodes".emRelations.em7.monitoring.UserDefine.StackRnR_SemiAuto )
   END_RUNG wire#w5
   RUNG wire#w2
      Contact( "Unit1.EmNodes".BA040.StackToReelCut.UnitStatus.specialFunctions.GaugeRnR3Cathode )
   END_RUNG wire#w7
   RUNG wire#powerrail
      Contact( "Unit1.EmNodes".emRelations.em7.monitoring.UserDefine.RunOut_SemiAuto )
   END_RUNG wire#w5
   // the same network as SCL:
   #statTonTimer[11].TON(IN := (((#statUnitStatus.state.execute OR #statUnitStatus.state.stopping OR #statUnitStatus.state.holding OR #statUnitStatus.state.suspending OR #statUnitStatus.state.completing) AND ((#unitStatus.specialFunctions.reWrokMode AND ("Unit1.EmNodes".emRelations.em7.monitoring.UserDefine.Motion_Step_Excute OR ("Unit1.EmNodes".emRelations.em7.monitoring.UserDefine."Stack#2_CV_Unuse" AND "Unit1.MotionNodes".PLCToMotion.Parameter.ReelCutMain.StepAuto.Stack2CVUnUse)) AND ("Unit1.EmData".PartData[1].Common.PartStatus <> 0)) OR (#unitStatus.specialFunctions.runOut AND NOT "Unit1.EmNodes".emRelations.em7.monitoring.UserDefine.RunOut_Complete) OR (#unitStatus.specialFunctions.gaugeRnR_Type3 AND "Unit1.EmNodes".emRelations.em7.monitoring.UserDefine.ConveyorEmptyCMD) OR (("Unit1.EmNodes".BA030.StackToReelCut.UnitStatus.specialFunctions.GaugeRnR1CathodeAlign OR "Unit1.EmNodes".BA030.StackToReelCut.UnitStatus.specialFunctions.GaugeRnR3Cathode) AND ("Unit1.EmData".PartData[9].Common.PartStatus = 0) AND "Unit1.EmNodes".emRelations.em7.monitoring.UserDefine.StackRnR_SemiAuto) OR (("Unit1.EmNodes".BA040.StackToReelCut.UnitStatus.specialFunctions.GaugeRnR1CathodeAlign OR "Unit1.EmNodes".BA040.StackToReelCut.UnitStatus.specialFunctions.GaugeRnR3Cathode) AND ("Unit1.EmData".PartData[17].Common.PartStatus = 0) AND "Unit1.EmNodes".emRelations.em7.monitoring.UserDefine.StackRnR_SemiAuto))) OR "Unit1.EmNodes".emRelations.em7.monitoring.UserDefine.RunOut_SemiAuto) AND #instWebGuidMotionSemiStepJob6.interlock AND ("Unit1.Em3.ControlNodes".webGuid.jobs.status.activeJobNumber = 0) AND NOT "Unit1.MotionNodes".MotionToPLC.Stauts.ReelCutMain.Busy,
                         PT := T#10ms);
   #_w1 := #statTonTimer[11].Q AND NOT #statPulse[0];   // rising edge
   #statPulse[0] := #statTonTimer[11].Q;
   #instWebGuidMotionSemiStepJob6(parentReferenceDesignator := "Unit1.Em3.Config".em.referenceDesignator.combined,   // "LAF_SelectJob"
                           jobNumber := "U1EM3_JOB06",
                           singleCycleJob := #FALSE,
                           interlock := NOT #statCheckCamRecipeChangedStatus.ExecuteRequired AND #statCheckCamRecipeChangedStatus.ValidParameters,
                           startCondition := #_w1,
                           hmiInterface := "Unit1.Em3.HmiInterface".webGuid.jobs,
                           jobs := "Unit1.Em3.ControlNodes".webGuid.jobs,
                           jobStatus => "Unit1.EmNodes".emRelations.em3.monitoring.Jobstatus.WebGuidMotionSemiStepJob6);
END_REGION

REGION Network 23: Select Job [7] Motion CycleStop
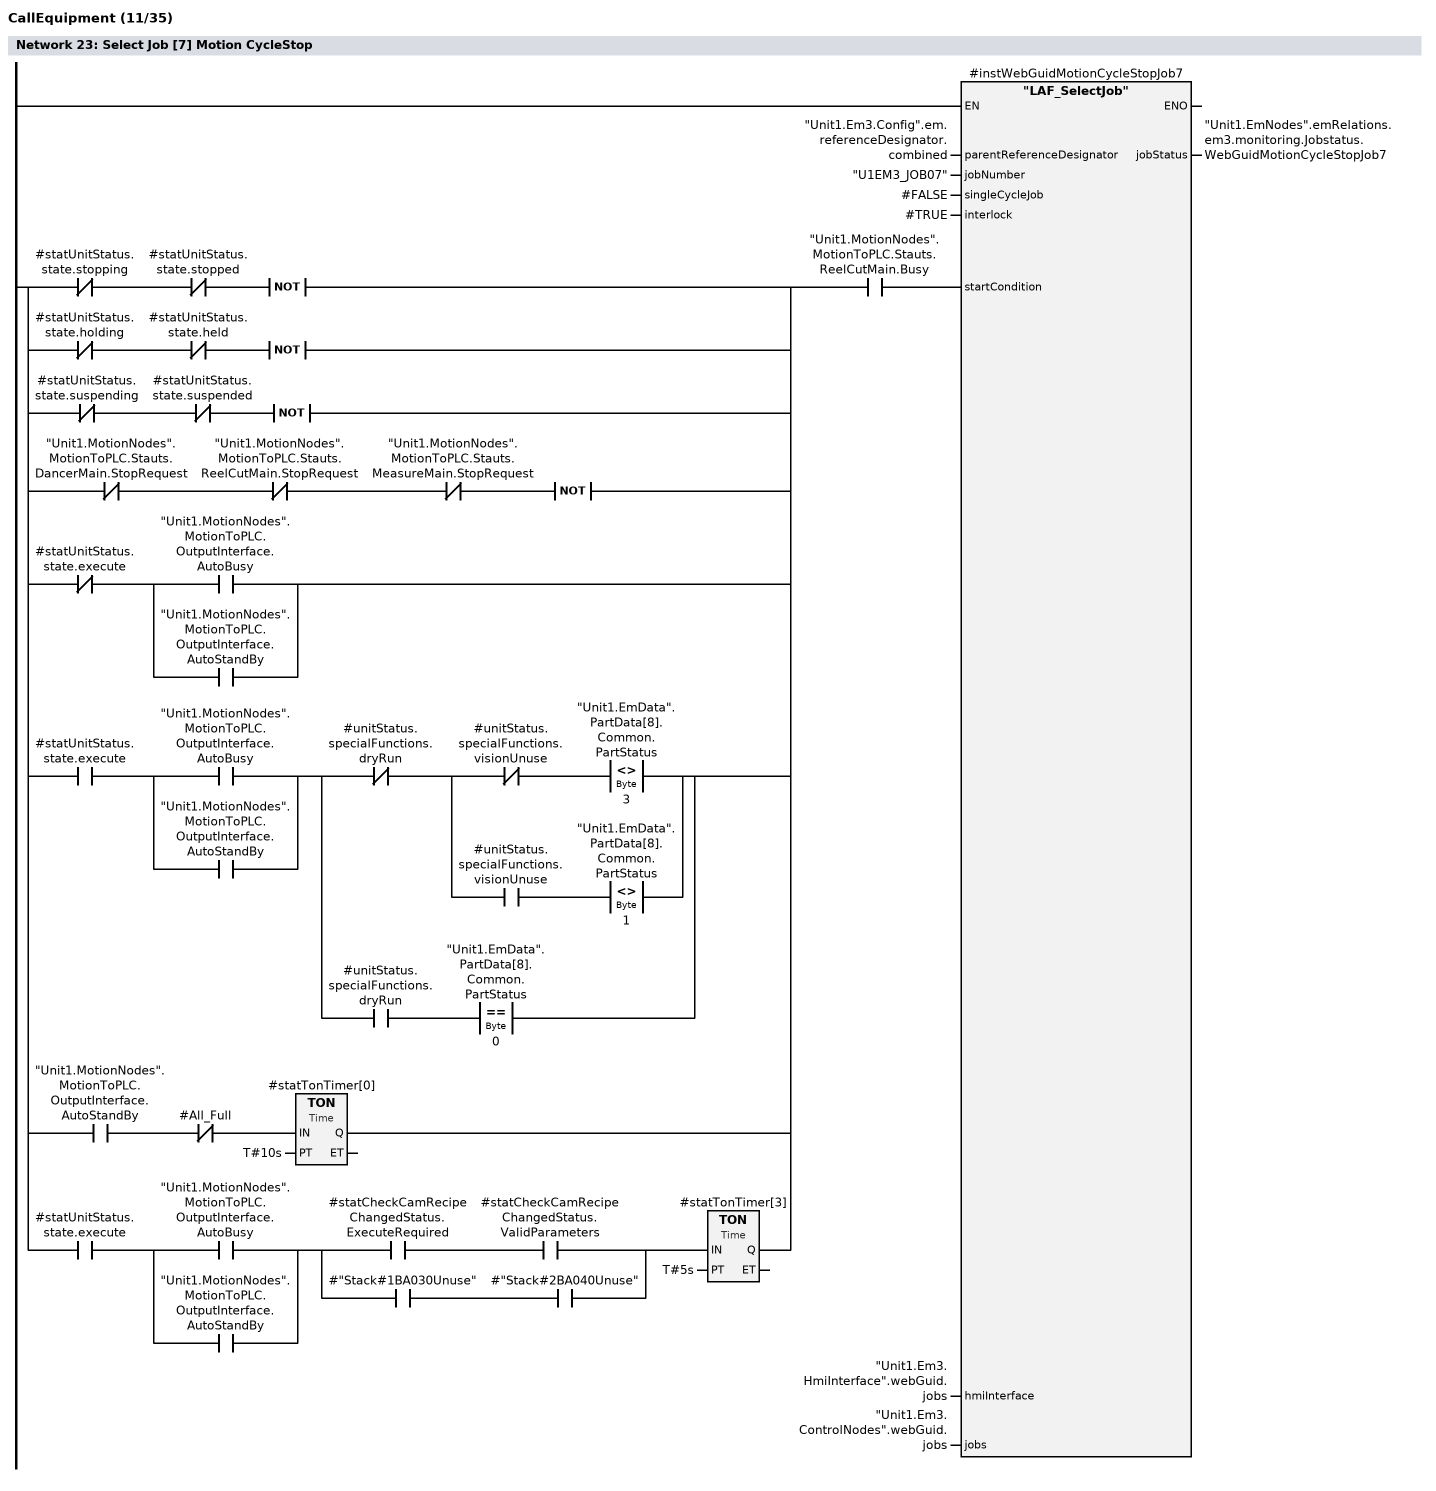
   RUNG wire#powerrail
      #instWebGuidMotionCycleStopJob7(startCondition := wire#w9, parentReferenceDesignator := "Unit1.Em3.Config".em.referenceDesignator.combined, jobNumber := "U1EM3_JOB07", singleCycleJob := #FALSE, interlock := #TRUE, hmiInterface := "Unit1.Em3.HmiInterface".webGuid.jobs, jobs := "Unit1.Em3.ControlNodes".webGuid.jobs, jobStatus => "Unit1.EmNodes".emRelations.em3.monitoring.Jobstatus.WebGuidMotionCycleStopJob7)
   END_RUNG
   RUNG wire#powerrail
      I_Contact( #statUnitStatus.state.stopping )
      I_Contact( #statUnitStatus.state.stopped )
      Not()
      wire#w1
      Contact( "Unit1.MotionNodes".MotionToPLC.Stauts.ReelCutMain.Busy )
   END_RUNG wire#w9
   RUNG wire#powerrail
      I_Contact( #statUnitStatus.state.holding )
      I_Contact( #statUnitStatus.state.held )
      Not()
   END_RUNG wire#w1
   RUNG wire#powerrail
      I_Contact( #statUnitStatus.state.suspending )
      I_Contact( #statUnitStatus.state.suspended )
      Not()
   END_RUNG wire#w1
   RUNG wire#powerrail
      I_Contact( "Unit1.MotionNodes".MotionToPLC.Stauts.DancerMain.StopRequest )
      I_Contact( "Unit1.MotionNodes".MotionToPLC.Stauts.ReelCutMain.StopRequest )
      I_Contact( "Unit1.MotionNodes".MotionToPLC.Stauts.MeasureMain.StopRequest )
      Not()
   END_RUNG wire#w1
   RUNG wire#powerrail
      I_Contact( #statUnitStatus.state.execute )
      wire#w2
      Contact( "Unit1.MotionNodes".MotionToPLC.OutputInterface.AutoBusy )
   END_RUNG wire#w1
   RUNG wire#w2
      Contact( "Unit1.MotionNodes".MotionToPLC.OutputInterface.AutoStandBy )
   END_RUNG wire#w1
   RUNG wire#powerrail
      Contact( #statUnitStatus.state.execute )
      wire#w3
      Contact( "Unit1.MotionNodes".MotionToPLC.OutputInterface.AutoBusy )
      wire#w4
      I_Contact( #unitStatus.specialFunctions.dryRun )
      wire#w5
      I_Contact( #unitStatus.specialFunctions.visionUnuse )
      { S7_Templates := "SrcType := Byte" } NE_Contact(in1 := "Unit1.EmData".PartData[8].Common.PartStatus, in2 := 3)
   END_RUNG wire#w1
   RUNG wire#w3
      Contact( "Unit1.MotionNodes".MotionToPLC.OutputInterface.AutoStandBy )
   END_RUNG wire#w4
   RUNG wire#w5
      Contact( #unitStatus.specialFunctions.visionUnuse )
      { S7_Templates := "SrcType := Byte" } NE_Contact(in1 := "Unit1.EmData".PartData[8].Common.PartStatus, in2 := 1)
   END_RUNG wire#w1
   RUNG wire#w4
      Contact( #unitStatus.specialFunctions.dryRun )
      { S7_Templates := "SrcType := Byte" } EQ_Contact(in1 := "Unit1.EmData".PartData[8].Common.PartStatus, in2 := 0)
   END_RUNG wire#w1
   RUNG wire#powerrail
      Contact( "Unit1.MotionNodes".MotionToPLC.OutputInterface.AutoStandBy )
      I_Contact( #All_Full )
      { S7_Templates := "time_type := Time" } #statTonTimer[0].TON(pt := T#10s, et =>)
   END_RUNG wire#w1
   RUNG wire#powerrail
      Contact( #statUnitStatus.state.execute )
      wire#w6
      Contact( "Unit1.MotionNodes".MotionToPLC.OutputInterface.AutoBusy )
      wire#w7
      Contact( #statCheckCamRecipeChangedStatus.ExecuteRequired )
      Contact( #statCheckCamRecipeChangedStatus.ValidParameters )
      wire#w8
      { S7_Templates := "time_type := Time" } #statTonTimer[3].TON(pt := T#5s, et =>)
   END_RUNG wire#w1
   RUNG wire#w6
      Contact( "Unit1.MotionNodes".MotionToPLC.OutputInterface.AutoStandBy )
   END_RUNG wire#w7
   RUNG wire#w7
      Contact( #"Stack#1BA030Unuse" )
      Contact( #"Stack#2BA040Unuse" )
   END_RUNG wire#w8
   // the same network as SCL:
   #statTonTimer[0].TON(IN := "Unit1.MotionNodes".MotionToPLC.OutputInterface.AutoStandBy AND NOT #All_Full,
                        PT := T#10s);
   #_w1 := #statTonTimer[0].Q;
   #statTonTimer[3].TON(IN := #statUnitStatus.state.execute AND ("Unit1.MotionNodes".MotionToPLC.OutputInterface.AutoBusy OR "Unit1.MotionNodes".MotionToPLC.OutputInterface.AutoStandBy) AND ((#statCheckCamRecipeChangedStatus.ExecuteRequired AND #statCheckCamRecipeChangedStatus.ValidParameters) OR (#"Stack#1BA030Unuse" AND #"Stack#2BA040Unuse")),
                        PT := T#5s);
   #instWebGuidMotionCycleStopJob7(parentReferenceDesignator := "Unit1.Em3.Config".em.referenceDesignator.combined,   // "LAF_SelectJob"
                           jobNumber := "U1EM3_JOB07",
                           singleCycleJob := #FALSE,
                           interlock := #TRUE,
                           startCondition := (NOT (NOT #statUnitStatus.state.stopping AND NOT #statUnitStatus.state.stopped) OR NOT (NOT #statUnitStatus.state.holding AND NOT #statUnitStatus.state.held) OR NOT (NOT #statUnitStatus.state.suspending AND NOT #statUnitStatus.state.suspended) OR NOT (NOT "Unit1.MotionNodes".MotionToPLC.Stauts.DancerMain.StopRequest AND NOT "Unit1.MotionNodes".MotionToPLC.Stauts.ReelCutMain.StopRequest AND NOT "Unit1.MotionNodes".MotionToPLC.Stauts.MeasureMain.StopRequest) OR (NOT #statUnitStatus.state.execute AND ("Unit1.MotionNodes".MotionToPLC.OutputInterface.AutoBusy OR "Unit1.MotionNodes".MotionToPLC.OutputInterface.AutoStandBy)) OR (#statUnitStatus.state.execute AND ("Unit1.MotionNodes".MotionToPLC.OutputInterface.AutoBusy OR "Unit1.MotionNodes".MotionToPLC.OutputInterface.AutoStandBy) AND ((NOT #unitStatus.specialFunctions.dryRun AND ((NOT #unitStatus.specialFunctions.visionUnuse AND ("Unit1.EmData".PartData[8].Common.PartStatus <> 3)) OR (#unitStatus.specialFunctions.visionUnuse AND ("Unit1.EmData".PartData[8].Common.PartStatus <> 1)))) OR (#unitStatus.specialFunctions.dryRun AND ("Unit1.EmData".PartData[8].Common.PartStatus = 0)))) OR #_w1 OR #statTonTimer[3].Q) AND "Unit1.MotionNodes".MotionToPLC.Stauts.ReelCutMain.Busy,
                           hmiInterface := "Unit1.Em3.HmiInterface".webGuid.jobs,
                           jobs := "Unit1.Em3.ControlNodes".webGuid.jobs,
                           jobStatus => "Unit1.EmNodes".emRelations.em3.monitoring.Jobstatus.WebGuidMotionCycleStopJob7);
END_REGION

REGION Network 24: Select Job [8] Motion FastStop
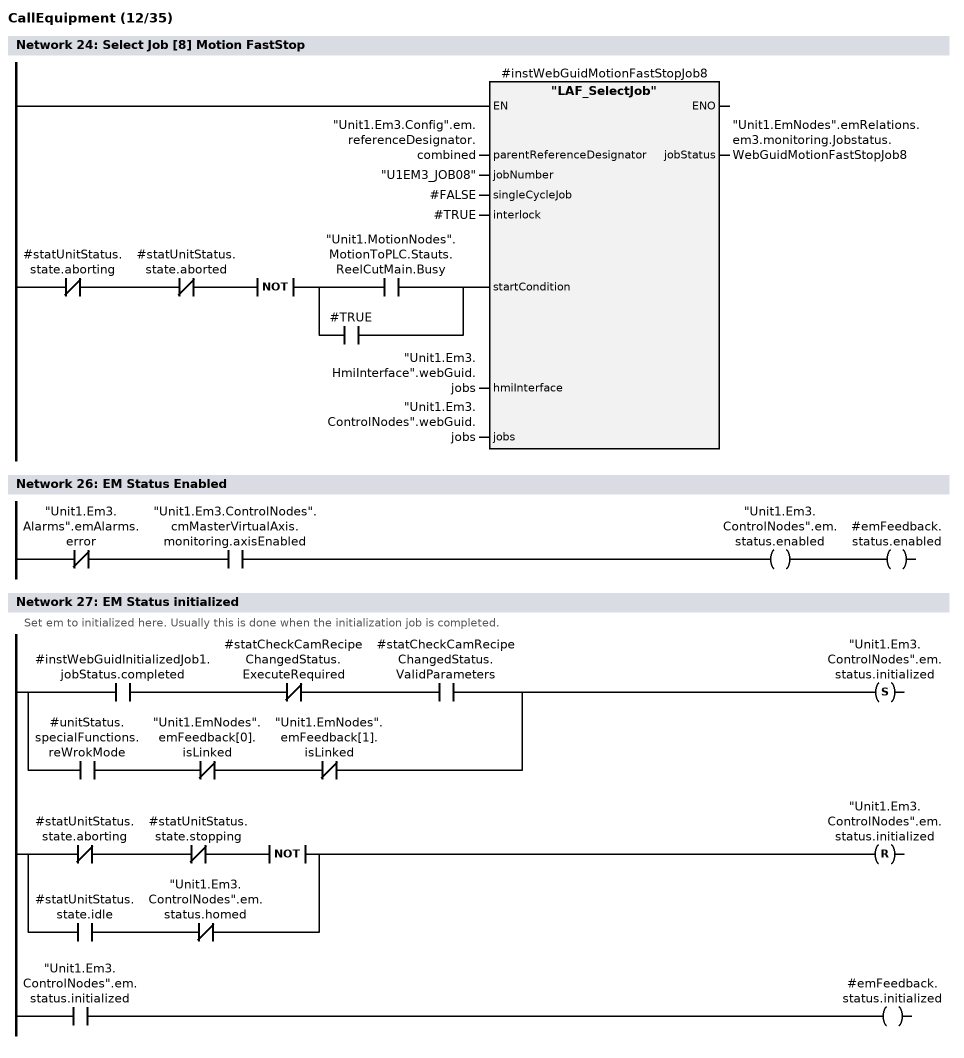
   RUNG wire#powerrail
      #instWebGuidMotionFastStopJob8(startCondition := wire#w2, parentReferenceDesignator := "Unit1.Em3.Config".em.referenceDesignator.combined, jobNumber := "U1EM3_JOB08", singleCycleJob := #FALSE, interlock := #TRUE, hmiInterface := "Unit1.Em3.HmiInterface".webGuid.jobs, jobs := "Unit1.Em3.ControlNodes".webGuid.jobs, jobStatus => "Unit1.EmNodes".emRelations.em3.monitoring.Jobstatus.WebGuidMotionFastStopJob8)
   END_RUNG
   RUNG wire#powerrail
      I_Contact( #statUnitStatus.state.aborting )
      I_Contact( #statUnitStatus.state.aborted )
      Not()
      wire#w1
      Contact( "Unit1.MotionNodes".MotionToPLC.Stauts.ReelCutMain.Busy )
   END_RUNG wire#w2
   RUNG wire#w1
      Contact( #TRUE )
   END_RUNG wire#w2
   // the same network as SCL:
   #instWebGuidMotionFastStopJob8(parentReferenceDesignator := "Unit1.Em3.Config".em.referenceDesignator.combined,   // "LAF_SelectJob"
                           jobNumber := "U1EM3_JOB08",
                           singleCycleJob := #FALSE,
                           interlock := #TRUE,
                           startCondition := NOT (NOT #statUnitStatus.state.aborting AND NOT #statUnitStatus.state.aborted) AND ("Unit1.MotionNodes".MotionToPLC.Stauts.ReelCutMain.Busy OR #TRUE),
                           hmiInterface := "Unit1.Em3.HmiInterface".webGuid.jobs,
                           jobs := "Unit1.Em3.ControlNodes".webGuid.jobs,
                           jobStatus => "Unit1.EmNodes".emRelations.em3.monitoring.Jobstatus.WebGuidMotionFastStopJob8);
END_REGION

REGION Network 25: WebGuid Job Working Done
END_REGION

REGION Network 26: EM Status Enabled
   RUNG wire#powerrail
      I_Contact( "Unit1.Em3.Alarms".emAlarms.error )
      Contact( "Unit1.Em3.ControlNodes".cmMasterVirtualAxis.monitoring.axisEnabled )
      Coil( "Unit1.Em3.ControlNodes".em.status.enabled )
      Coil( #emFeedback.status.enabled )
   END_RUNG
   // the same network as SCL:
   "Unit1.Em3.ControlNodes".em.status.enabled := NOT "Unit1.Em3.Alarms".emAlarms.error AND "Unit1.Em3.ControlNodes".cmMasterVirtualAxis.monitoring.axisEnabled;
   #emFeedback.status.enabled := "Unit1.Em3.ControlNodes".em.status.enabled;
END_REGION

REGION Network 27: EM Status initialized
   // Set em to initialized here. Usually this is done when the initialization job is completed.
   RUNG wire#powerrail
      Contact( #instWebGuidInitializedJob1.jobStatus.completed )
      I_Contact( #statCheckCamRecipeChangedStatus.ExecuteRequired )
      Contact( #statCheckCamRecipeChangedStatus.ValidParameters )
      wire#w1
      S_Coil( "Unit1.Em3.ControlNodes".em.status.initialized )
   END_RUNG
   RUNG wire#powerrail
      Contact( #unitStatus.specialFunctions.reWrokMode )
      I_Contact( "Unit1.EmNodes".emFeedback[0].isLinked )
      I_Contact( "Unit1.EmNodes".emFeedback[1].isLinked )
   END_RUNG wire#w1
   RUNG wire#powerrail
      I_Contact( #statUnitStatus.state.aborting )
      I_Contact( #statUnitStatus.state.stopping )
      Not()
      wire#w2
      R_Coil( "Unit1.Em3.ControlNodes".em.status.initialized )
   END_RUNG
   RUNG wire#powerrail
      Contact( #statUnitStatus.state.idle )
      I_Contact( "Unit1.Em3.ControlNodes".em.status.homed )
   END_RUNG wire#w2
   RUNG wire#powerrail
      Contact( "Unit1.Em3.ControlNodes".em.status.initialized )
      Coil( #emFeedback.status.initialized )
   END_RUNG
   // the same network as SCL:
   IF (#instWebGuidInitializedJob1.jobStatus.completed AND NOT #statCheckCamRecipeChangedStatus.ExecuteRequired AND #statCheckCamRecipeChangedStatus.ValidParameters) OR (#unitStatus.specialFunctions.reWrokMode AND NOT "Unit1.EmNodes".emFeedback[0].isLinked AND NOT "Unit1.EmNodes".emFeedback[1].isLinked) THEN
       "Unit1.Em3.ControlNodes".em.status.initialized := TRUE;
   END_IF;
   IF NOT (NOT #statUnitStatus.state.aborting AND NOT #statUnitStatus.state.stopping) OR (#statUnitStatus.state.idle AND NOT "Unit1.Em3.ControlNodes".em.status.homed) THEN
       "Unit1.Em3.ControlNodes".em.status.initialized := FALSE;
   END_IF;
   #emFeedback.status.initialized := "Unit1.Em3.ControlNodes".em.status.initialized;
END_REGION

REGION Network 28: EM Status Homed
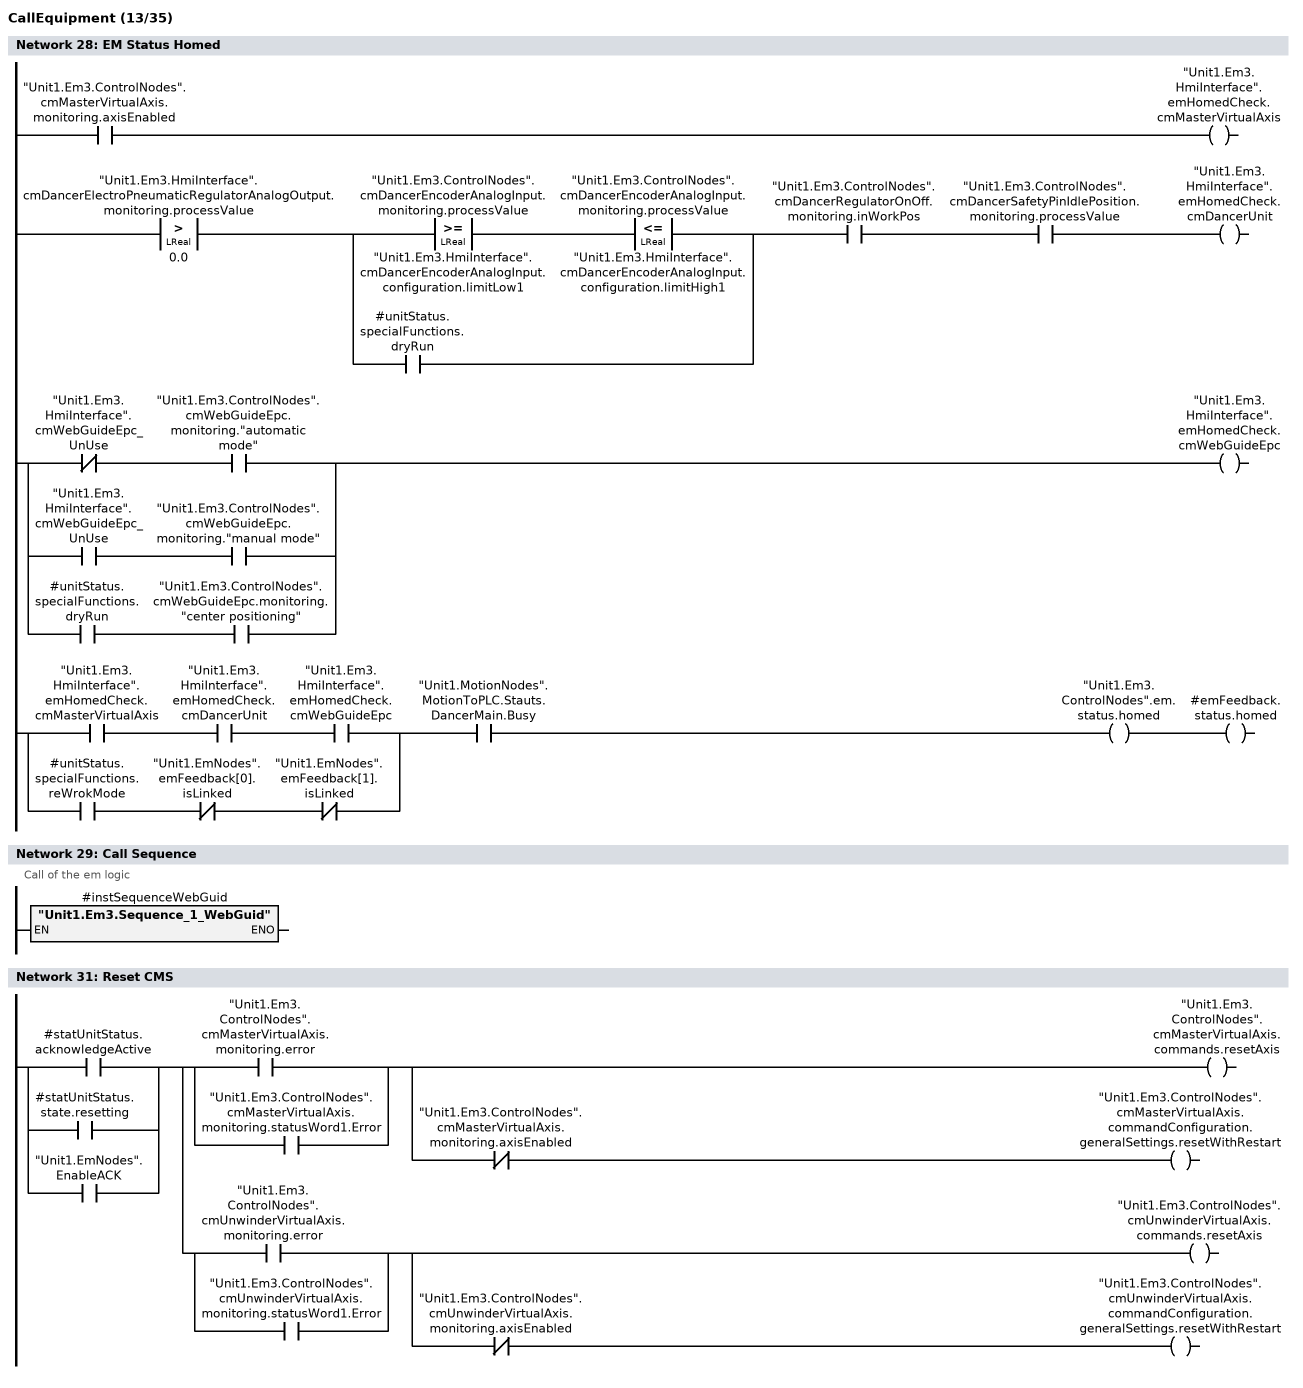
   RUNG wire#powerrail
      Contact( "Unit1.Em3.ControlNodes".cmMasterVirtualAxis.monitoring.axisEnabled )
      Coil( "Unit1.Em3.HmiInterface".emHomedCheck.cmMasterVirtualAxis )
   END_RUNG
   RUNG wire#powerrail
      { S7_Templates := "SrcType := LReal" } GT_Contact(in1 := "Unit1.Em3.HmiInterface".cmDancerElectroPneumaticRegulatorAnalogOutput.monitoring.processValue, in2 := 0.0)
      wire#w1
      { S7_Templates := "SrcType := LReal" } GE_Contact(in1 := "Unit1.Em3.ControlNodes".cmDancerEncoderAnalogInput.monitoring.processValue, in2 := "Unit1.Em3.HmiInterface".cmDancerEncoderAnalogInput.configuration.limitLow1)
      { S7_Templates := "SrcType := LReal" } LE_Contact(in1 := "Unit1.Em3.ControlNodes".cmDancerEncoderAnalogInput.monitoring.processValue, in2 := "Unit1.Em3.HmiInterface".cmDancerEncoderAnalogInput.configuration.limitHigh1)
      wire#w2
      Contact( "Unit1.Em3.ControlNodes".cmDancerRegulatorOnOff.monitoring.inWorkPos )
      Contact( "Unit1.Em3.ControlNodes".cmDancerSafetyPinIdlePosition.monitoring.processValue )
      Coil( "Unit1.Em3.HmiInterface".emHomedCheck.cmDancerUnit )
   END_RUNG
   RUNG wire#w1
      Contact( #unitStatus.specialFunctions.dryRun )
   END_RUNG wire#w2
   RUNG wire#powerrail
      I_Contact( "Unit1.Em3.HmiInterface".cmWebGuideEpc_UnUse )
      Contact( "Unit1.Em3.ControlNodes".cmWebGuideEpc.monitoring."automatic mode" )
      wire#w3
      Coil( "Unit1.Em3.HmiInterface".emHomedCheck.cmWebGuideEpc )
   END_RUNG
   RUNG wire#powerrail
      Contact( "Unit1.Em3.HmiInterface".cmWebGuideEpc_UnUse )
      Contact( "Unit1.Em3.ControlNodes".cmWebGuideEpc.monitoring."manual mode" )
   END_RUNG wire#w3
   RUNG wire#powerrail
      Contact( #unitStatus.specialFunctions.dryRun )
      Contact( "Unit1.Em3.ControlNodes".cmWebGuideEpc.monitoring."center positioning" )
   END_RUNG wire#w3
   RUNG wire#powerrail
      Contact( "Unit1.Em3.HmiInterface".emHomedCheck.cmMasterVirtualAxis )
      Contact( "Unit1.Em3.HmiInterface".emHomedCheck.cmDancerUnit )
      Contact( "Unit1.Em3.HmiInterface".emHomedCheck.cmWebGuideEpc )
      wire#w4
      Contact( "Unit1.MotionNodes".MotionToPLC.Stauts.DancerMain.Busy )
      Coil( "Unit1.Em3.ControlNodes".em.status.homed )
      Coil( #emFeedback.status.homed )
   END_RUNG
   RUNG wire#powerrail
      Contact( #unitStatus.specialFunctions.reWrokMode )
      I_Contact( "Unit1.EmNodes".emFeedback[0].isLinked )
      I_Contact( "Unit1.EmNodes".emFeedback[1].isLinked )
   END_RUNG wire#w4
   // the same network as SCL:
   "Unit1.Em3.HmiInterface".emHomedCheck.cmMasterVirtualAxis := "Unit1.Em3.ControlNodes".cmMasterVirtualAxis.monitoring.axisEnabled;
   "Unit1.Em3.HmiInterface".emHomedCheck.cmDancerUnit := ("Unit1.Em3.HmiInterface".cmDancerElectroPneumaticRegulatorAnalogOutput.monitoring.processValue > 0.0) AND ((("Unit1.Em3.ControlNodes".cmDancerEncoderAnalogInput.monitoring.processValue >= "Unit1.Em3.HmiInterface".cmDancerEncoderAnalogInput.configuration.limitLow1) AND ("Unit1.Em3.ControlNodes".cmDancerEncoderAnalogInput.monitoring.processValue <= "Unit1.Em3.HmiInterface".cmDancerEncoderAnalogInput.configuration.limitHigh1)) OR #unitStatus.specialFunctions.dryRun) AND "Unit1.Em3.ControlNodes".cmDancerRegulatorOnOff.monitoring.inWorkPos AND "Unit1.Em3.ControlNodes".cmDancerSafetyPinIdlePosition.monitoring.processValue;
   "Unit1.Em3.HmiInterface".emHomedCheck.cmWebGuideEpc := (NOT "Unit1.Em3.HmiInterface".cmWebGuideEpc_UnUse AND "Unit1.Em3.ControlNodes".cmWebGuideEpc.monitoring."automatic mode") OR ("Unit1.Em3.HmiInterface".cmWebGuideEpc_UnUse AND "Unit1.Em3.ControlNodes".cmWebGuideEpc.monitoring."manual mode") OR (#unitStatus.specialFunctions.dryRun AND "Unit1.Em3.ControlNodes".cmWebGuideEpc.monitoring."center positioning");
   "Unit1.Em3.ControlNodes".em.status.homed := (("Unit1.Em3.HmiInterface".emHomedCheck.cmMasterVirtualAxis AND "Unit1.Em3.HmiInterface".emHomedCheck.cmDancerUnit AND "Unit1.Em3.HmiInterface".emHomedCheck.cmWebGuideEpc) OR (#unitStatus.specialFunctions.reWrokMode AND NOT "Unit1.EmNodes".emFeedback[0].isLinked AND NOT "Unit1.EmNodes".emFeedback[1].isLinked)) AND "Unit1.MotionNodes".MotionToPLC.Stauts.DancerMain.Busy;
   #emFeedback.status.homed := "Unit1.Em3.ControlNodes".em.status.homed;
END_REGION

REGION Network 29: Call Sequence
   // Call of the em logic
   RUNG wire#powerrail
      #instSequenceWebGuid()
   END_RUNG
   // the same network as SCL:
   #instSequenceWebGuid();   // "Unit1.Em3.Sequence_1_WebGuid"
END_REGION

REGION Network 30: ******************** Control Modules (Axis) ********************
   // Call control modules that are actuators after the em logic (jobs and sequence), so that the latest commands are applied to the actuators.
END_REGION

REGION Network 31: Reset CMS
   RUNG wire#powerrail
      Contact( #statUnitStatus.acknowledgeActive )
      wire#w1
      Contact( "Unit1.Em3.ControlNodes".cmMasterVirtualAxis.monitoring.error )
      wire#w2
      Coil( "Unit1.Em3.ControlNodes".cmMasterVirtualAxis.commands.resetAxis )
   END_RUNG
   RUNG wire#powerrail
      Contact( #statUnitStatus.state.resetting )
   END_RUNG wire#w1
   RUNG wire#powerrail
      Contact( "Unit1.EmNodes".EnableACK )
   END_RUNG wire#w1
   RUNG wire#w1
      Contact( "Unit1.Em3.ControlNodes".cmMasterVirtualAxis.monitoring.statusWord1.Error )
   END_RUNG wire#w2
   RUNG wire#w2
      I_Contact( "Unit1.Em3.ControlNodes".cmMasterVirtualAxis.monitoring.axisEnabled )
      Coil( "Unit1.Em3.ControlNodes".cmMasterVirtualAxis.commandConfiguration.generalSettings.resetWithRestart )
   END_RUNG
   RUNG wire#w1
      Contact( "Unit1.Em3.ControlNodes".cmUnwinderVirtualAxis.monitoring.error )
      wire#w3
      Coil( "Unit1.Em3.ControlNodes".cmUnwinderVirtualAxis.commands.resetAxis )
   END_RUNG
   RUNG wire#w1
      Contact( "Unit1.Em3.ControlNodes".cmUnwinderVirtualAxis.monitoring.statusWord1.Error )
   END_RUNG wire#w3
   RUNG wire#w3
      I_Contact( "Unit1.Em3.ControlNodes".cmUnwinderVirtualAxis.monitoring.axisEnabled )
      Coil( "Unit1.Em3.ControlNodes".cmUnwinderVirtualAxis.commandConfiguration.generalSettings.resetWithRestart )
   END_RUNG
   // the same network as SCL:
   #_w1 := #statUnitStatus.acknowledgeActive OR #statUnitStatus.state.resetting OR "Unit1.EmNodes".EnableACK;
   "Unit1.Em3.ControlNodes".cmMasterVirtualAxis.commands.resetAxis := #_w1 AND ("Unit1.Em3.ControlNodes".cmMasterVirtualAxis.monitoring.error OR "Unit1.Em3.ControlNodes".cmMasterVirtualAxis.monitoring.statusWord1.Error);
   "Unit1.Em3.ControlNodes".cmMasterVirtualAxis.commandConfiguration.generalSettings.resetWithRestart := "Unit1.Em3.ControlNodes".cmMasterVirtualAxis.commands.resetAxis AND NOT "Unit1.Em3.ControlNodes".cmMasterVirtualAxis.monitoring.axisEnabled;
   "Unit1.Em3.ControlNodes".cmUnwinderVirtualAxis.commands.resetAxis := #_w1 AND ("Unit1.Em3.ControlNodes".cmUnwinderVirtualAxis.monitoring.error OR "Unit1.Em3.ControlNodes".cmUnwinderVirtualAxis.monitoring.statusWord1.Error);
   "Unit1.Em3.ControlNodes".cmUnwinderVirtualAxis.commandConfiguration.generalSettings.resetWithRestart := "Unit1.Em3.ControlNodes".cmUnwinderVirtualAxis.commands.resetAxis AND NOT "Unit1.Em3.ControlNodes".cmUnwinderVirtualAxis.monitoring.axisEnabled;
END_REGION

REGION Network 32: Enable/Disable CMs
   // Enable the axis during the resetting state and disable the axis during the aborting state.
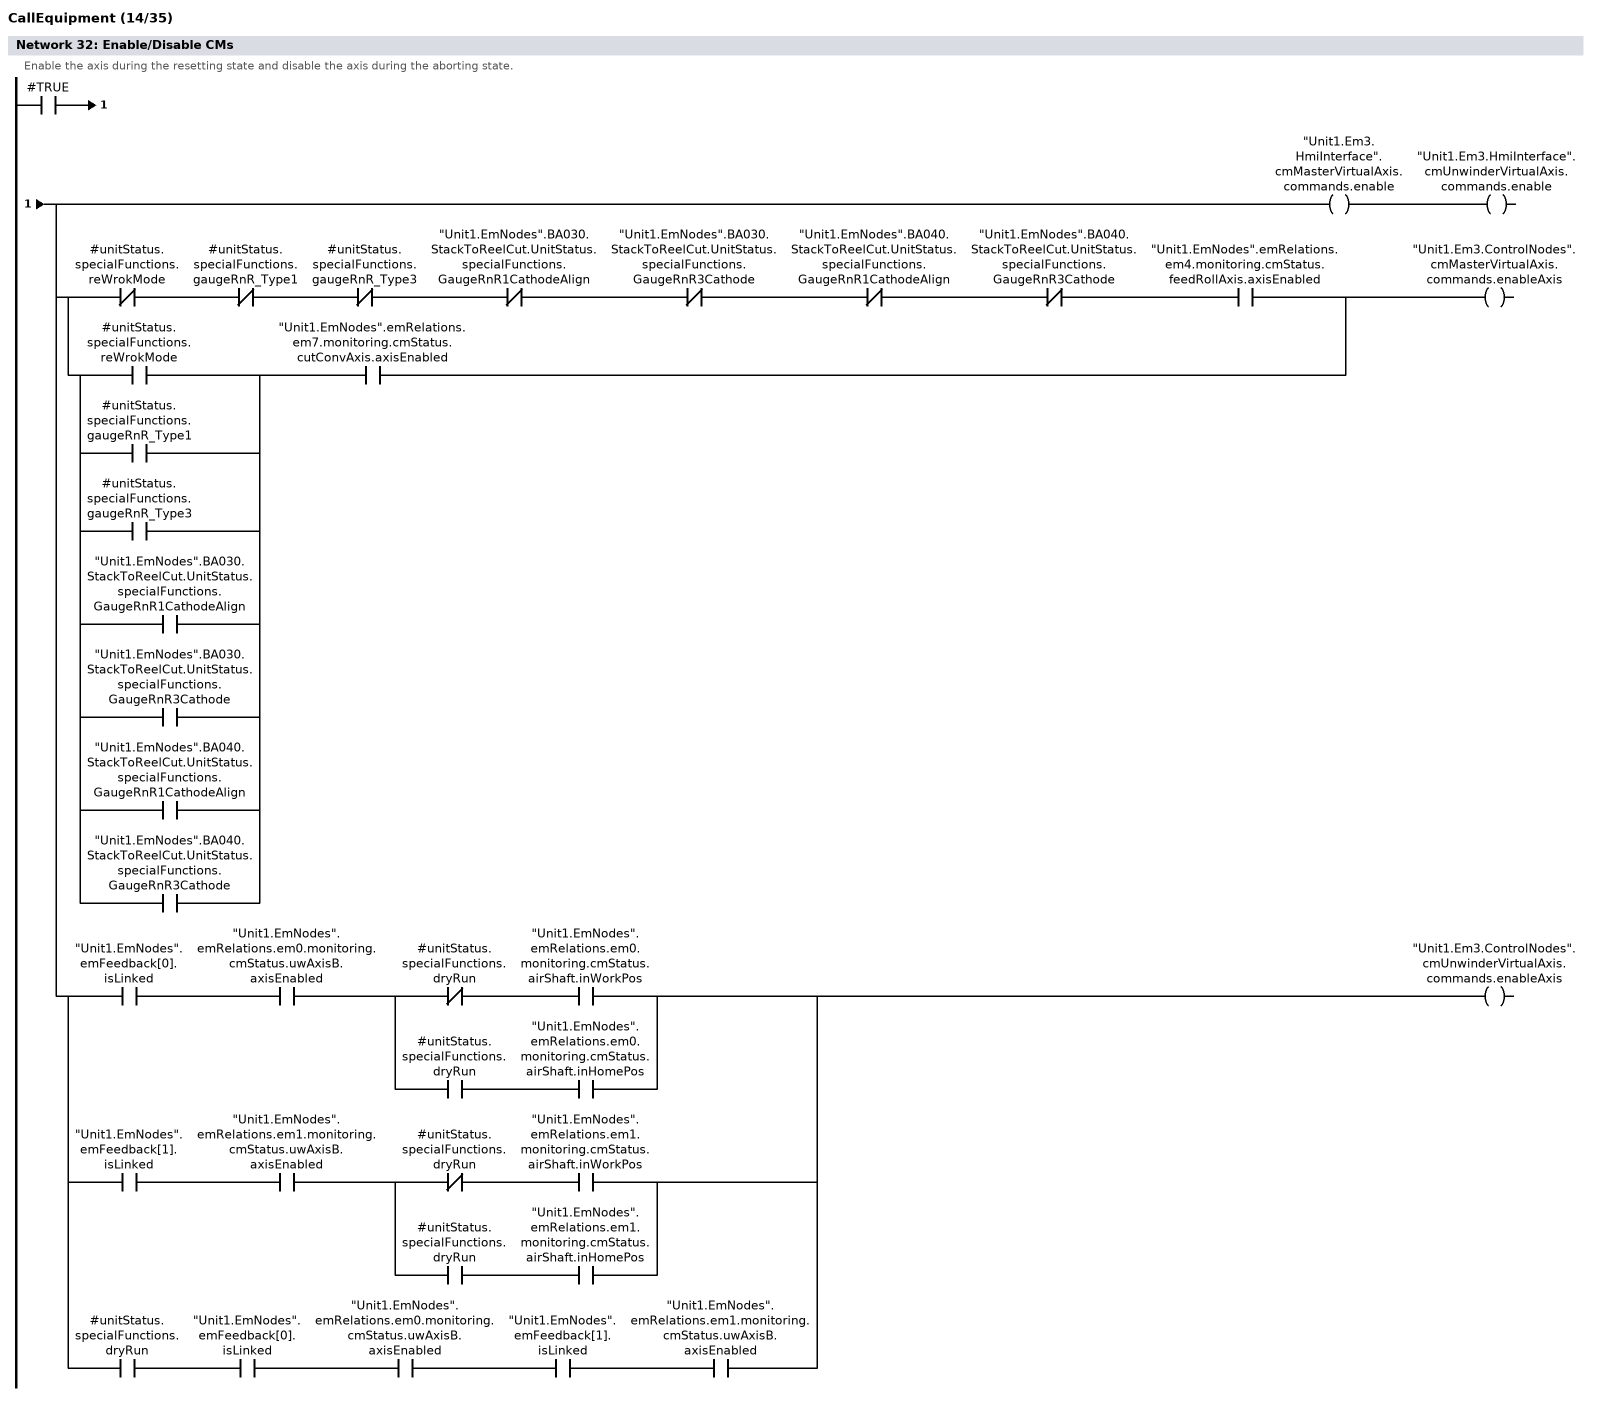
   RUNG wire#powerrail
      Contact( #TRUE )
      wire#w1
      Coil( "Unit1.Em3.HmiInterface".cmMasterVirtualAxis.commands.enable )
      Coil( "Unit1.Em3.HmiInterface".cmUnwinderVirtualAxis.commands.enable )
   END_RUNG
   RUNG wire#w1
      I_Contact( #unitStatus.specialFunctions.reWrokMode )
      I_Contact( #unitStatus.specialFunctions.gaugeRnR_Type1 )
      I_Contact( #unitStatus.specialFunctions.gaugeRnR_Type3 )
      I_Contact( "Unit1.EmNodes".BA030.StackToReelCut.UnitStatus.specialFunctions.GaugeRnR1CathodeAlign )
      I_Contact( "Unit1.EmNodes".BA030.StackToReelCut.UnitStatus.specialFunctions.GaugeRnR3Cathode )
      I_Contact( "Unit1.EmNodes".BA040.StackToReelCut.UnitStatus.specialFunctions.GaugeRnR1CathodeAlign )
      I_Contact( "Unit1.EmNodes".BA040.StackToReelCut.UnitStatus.specialFunctions.GaugeRnR3Cathode )
      Contact( "Unit1.EmNodes".emRelations.em4.monitoring.cmStatus.feedRollAxis.axisEnabled )
      wire#w2
      Coil( "Unit1.Em3.ControlNodes".cmMasterVirtualAxis.commands.enableAxis )
   END_RUNG
   RUNG wire#w1
      Contact( #unitStatus.specialFunctions.reWrokMode )
      wire#w3
      Contact( "Unit1.EmNodes".emRelations.em7.monitoring.cmStatus.cutConvAxis.axisEnabled )
   END_RUNG wire#w2
   RUNG wire#w1
      Contact( #unitStatus.specialFunctions.gaugeRnR_Type1 )
   END_RUNG wire#w3
   RUNG wire#w1
      Contact( #unitStatus.specialFunctions.gaugeRnR_Type3 )
   END_RUNG wire#w3
   RUNG wire#w1
      Contact( "Unit1.EmNodes".BA030.StackToReelCut.UnitStatus.specialFunctions.GaugeRnR1CathodeAlign )
   END_RUNG wire#w3
   RUNG wire#w1
      Contact( "Unit1.EmNodes".BA030.StackToReelCut.UnitStatus.specialFunctions.GaugeRnR3Cathode )
   END_RUNG wire#w3
   RUNG wire#w1
      Contact( "Unit1.EmNodes".BA040.StackToReelCut.UnitStatus.specialFunctions.GaugeRnR1CathodeAlign )
   END_RUNG wire#w3
   RUNG wire#w1
      Contact( "Unit1.EmNodes".BA040.StackToReelCut.UnitStatus.specialFunctions.GaugeRnR3Cathode )
   END_RUNG wire#w3
   RUNG wire#w1
      Contact( "Unit1.EmNodes".emFeedback[0].isLinked )
      Contact( "Unit1.EmNodes".emRelations.em0.monitoring.cmStatus.uwAxisB.axisEnabled )
      wire#w4
      I_Contact( #unitStatus.specialFunctions.dryRun )
      Contact( "Unit1.EmNodes".emRelations.em0.monitoring.cmStatus.airShaft.inWorkPos )
      wire#w5
      Coil( "Unit1.Em3.ControlNodes".cmUnwinderVirtualAxis.commands.enableAxis )
   END_RUNG
   RUNG wire#w4
      Contact( #unitStatus.specialFunctions.dryRun )
      Contact( "Unit1.EmNodes".emRelations.em0.monitoring.cmStatus.airShaft.inHomePos )
   END_RUNG wire#w5
   RUNG wire#w1
      Contact( "Unit1.EmNodes".emFeedback[1].isLinked )
      Contact( "Unit1.EmNodes".emRelations.em1.monitoring.cmStatus.uwAxisB.axisEnabled )
      wire#w6
      I_Contact( #unitStatus.specialFunctions.dryRun )
      Contact( "Unit1.EmNodes".emRelations.em1.monitoring.cmStatus.airShaft.inWorkPos )
   END_RUNG wire#w5
   RUNG wire#w6
      Contact( #unitStatus.specialFunctions.dryRun )
      Contact( "Unit1.EmNodes".emRelations.em1.monitoring.cmStatus.airShaft.inHomePos )
   END_RUNG wire#w5
   RUNG wire#w1
      Contact( #unitStatus.specialFunctions.dryRun )
      Contact( "Unit1.EmNodes".emFeedback[0].isLinked )
      Contact( "Unit1.EmNodes".emRelations.em0.monitoring.cmStatus.uwAxisB.axisEnabled )
      Contact( "Unit1.EmNodes".emFeedback[1].isLinked )
      Contact( "Unit1.EmNodes".emRelations.em1.monitoring.cmStatus.uwAxisB.axisEnabled )
   END_RUNG wire#w5
   // the same network as SCL:
   "Unit1.Em3.HmiInterface".cmMasterVirtualAxis.commands.enable := #TRUE;
   "Unit1.Em3.HmiInterface".cmUnwinderVirtualAxis.commands.enable := #TRUE;
   "Unit1.Em3.ControlNodes".cmMasterVirtualAxis.commands.enableAxis := #TRUE AND ((NOT #unitStatus.specialFunctions.reWrokMode AND NOT #unitStatus.specialFunctions.gaugeRnR_Type1 AND NOT #unitStatus.specialFunctions.gaugeRnR_Type3 AND NOT "Unit1.EmNodes".BA030.StackToReelCut.UnitStatus.specialFunctions.GaugeRnR1CathodeAlign AND NOT "Unit1.EmNodes".BA030.StackToReelCut.UnitStatus.specialFunctions.GaugeRnR3Cathode AND NOT "Unit1.EmNodes".BA040.StackToReelCut.UnitStatus.specialFunctions.GaugeRnR1CathodeAlign AND NOT "Unit1.EmNodes".BA040.StackToReelCut.UnitStatus.specialFunctions.GaugeRnR3Cathode AND "Unit1.EmNodes".emRelations.em4.monitoring.cmStatus.feedRollAxis.axisEnabled) OR ((#unitStatus.specialFunctions.reWrokMode OR #unitStatus.specialFunctions.gaugeRnR_Type1 OR #unitStatus.specialFunctions.gaugeRnR_Type3 OR "Unit1.EmNodes".BA030.StackToReelCut.UnitStatus.specialFunctions.GaugeRnR1CathodeAlign OR "Unit1.EmNodes".BA030.StackToReelCut.UnitStatus.specialFunctions.GaugeRnR3Cathode OR "Unit1.EmNodes".BA040.StackToReelCut.UnitStatus.specialFunctions.GaugeRnR1CathodeAlign OR "Unit1.EmNodes".BA040.StackToReelCut.UnitStatus.specialFunctions.GaugeRnR3Cathode) AND "Unit1.EmNodes".emRelations.em7.monitoring.cmStatus.cutConvAxis.axisEnabled));
   "Unit1.Em3.ControlNodes".cmUnwinderVirtualAxis.commands.enableAxis := #TRUE AND (("Unit1.EmNodes".emFeedback[0].isLinked AND "Unit1.EmNodes".emRelations.em0.monitoring.cmStatus.uwAxisB.axisEnabled AND ((NOT #unitStatus.specialFunctions.dryRun AND "Unit1.EmNodes".emRelations.em0.monitoring.cmStatus.airShaft.inWorkPos) OR (#unitStatus.specialFunctions.dryRun AND "Unit1.EmNodes".emRelations.em0.monitoring.cmStatus.airShaft.inHomePos))) OR ("Unit1.EmNodes".emFeedback[1].isLinked AND "Unit1.EmNodes".emRelations.em1.monitoring.cmStatus.uwAxisB.axisEnabled AND ((NOT #unitStatus.specialFunctions.dryRun AND "Unit1.EmNodes".emRelations.em1.monitoring.cmStatus.airShaft.inWorkPos) OR (#unitStatus.specialFunctions.dryRun AND "Unit1.EmNodes".emRelations.em1.monitoring.cmStatus.airShaft.inHomePos))) OR (#unitStatus.specialFunctions.dryRun AND "Unit1.EmNodes".emFeedback[0].isLinked AND "Unit1.EmNodes".emRelations.em0.monitoring.cmStatus.uwAxisB.axisEnabled AND "Unit1.EmNodes".emFeedback[1].isLinked AND "Unit1.EmNodes".emRelations.em1.monitoring.cmStatus.uwAxisB.axisEnabled));
END_REGION

REGION Network 33: CM Master Virtual Axis Command Jog
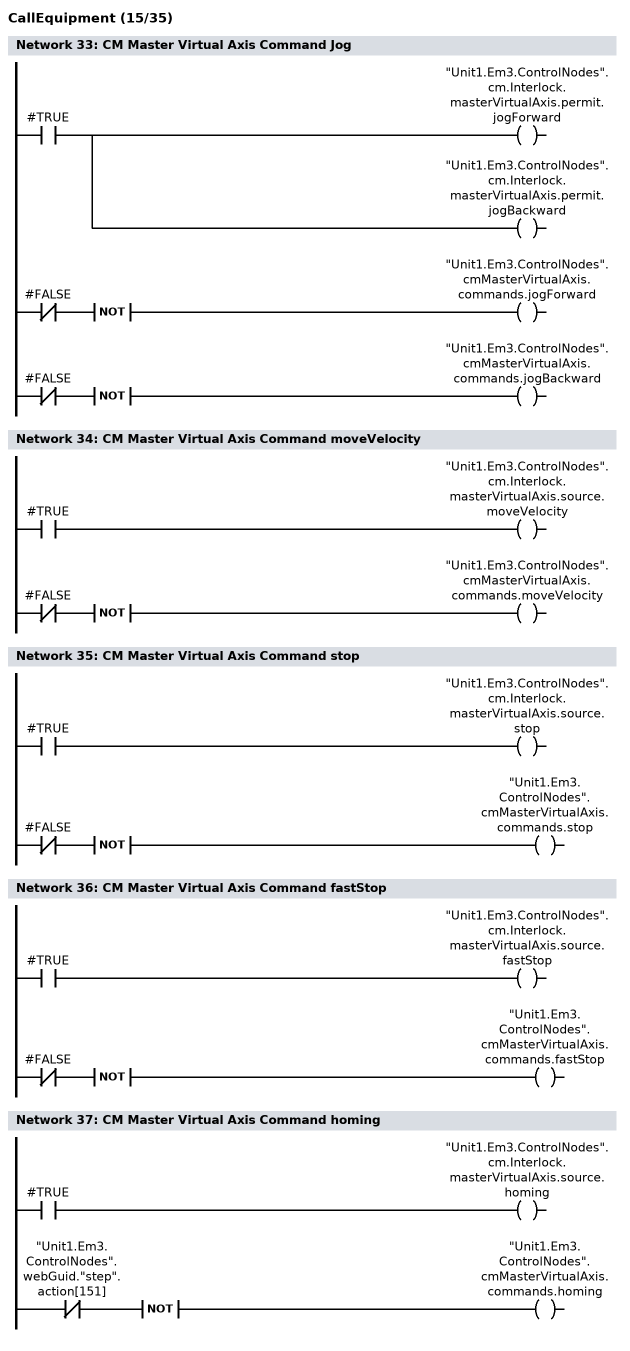
   RUNG wire#powerrail
      Contact( #TRUE )
      wire#w1
      Coil( "Unit1.Em3.ControlNodes".cm.Interlock.masterVirtualAxis.permit.jogForward )
   END_RUNG
   RUNG wire#w1
      Coil( "Unit1.Em3.ControlNodes".cm.Interlock.masterVirtualAxis.permit.jogBackward )
   END_RUNG
   RUNG wire#powerrail
      I_Contact( #FALSE )
      Not()
      Coil( "Unit1.Em3.ControlNodes".cmMasterVirtualAxis.commands.jogForward )
   END_RUNG
   RUNG wire#powerrail
      I_Contact( #FALSE )
      Not()
      Coil( "Unit1.Em3.ControlNodes".cmMasterVirtualAxis.commands.jogBackward )
   END_RUNG
   // the same network as SCL:
   "Unit1.Em3.ControlNodes".cm.Interlock.masterVirtualAxis.permit.jogForward := #TRUE;
   "Unit1.Em3.ControlNodes".cm.Interlock.masterVirtualAxis.permit.jogBackward := #TRUE;
   "Unit1.Em3.ControlNodes".cmMasterVirtualAxis.commands.jogForward := NOT (NOT #FALSE);
   "Unit1.Em3.ControlNodes".cmMasterVirtualAxis.commands.jogBackward := NOT (NOT #FALSE);
END_REGION

REGION Network 34: CM Master Virtual Axis Command moveVelocity
   RUNG wire#powerrail
      Contact( #TRUE )
      Coil( "Unit1.Em3.ControlNodes".cm.Interlock.masterVirtualAxis.source.moveVelocity )
   END_RUNG
   RUNG wire#powerrail
      I_Contact( #FALSE )
      Not()
      Coil( "Unit1.Em3.ControlNodes".cmMasterVirtualAxis.commands.moveVelocity )
   END_RUNG
   // the same network as SCL:
   "Unit1.Em3.ControlNodes".cm.Interlock.masterVirtualAxis.source.moveVelocity := #TRUE;
   "Unit1.Em3.ControlNodes".cmMasterVirtualAxis.commands.moveVelocity := NOT (NOT #FALSE);
END_REGION

REGION Network 35: CM Master Virtual Axis Command stop
   RUNG wire#powerrail
      Contact( #TRUE )
      Coil( "Unit1.Em3.ControlNodes".cm.Interlock.masterVirtualAxis.source.stop )
   END_RUNG
   RUNG wire#powerrail
      I_Contact( #FALSE )
      Not()
      Coil( "Unit1.Em3.ControlNodes".cmMasterVirtualAxis.commands.stop )
   END_RUNG
   // the same network as SCL:
   "Unit1.Em3.ControlNodes".cm.Interlock.masterVirtualAxis.source.stop := #TRUE;
   "Unit1.Em3.ControlNodes".cmMasterVirtualAxis.commands.stop := NOT (NOT #FALSE);
END_REGION

REGION Network 36: CM Master Virtual Axis Command fastStop
   RUNG wire#powerrail
      Contact( #TRUE )
      Coil( "Unit1.Em3.ControlNodes".cm.Interlock.masterVirtualAxis.source.fastStop )
   END_RUNG
   RUNG wire#powerrail
      I_Contact( #FALSE )
      Not()
      Coil( "Unit1.Em3.ControlNodes".cmMasterVirtualAxis.commands.fastStop )
   END_RUNG
   // the same network as SCL:
   "Unit1.Em3.ControlNodes".cm.Interlock.masterVirtualAxis.source.fastStop := #TRUE;
   "Unit1.Em3.ControlNodes".cmMasterVirtualAxis.commands.fastStop := NOT (NOT #FALSE);
END_REGION

REGION Network 37: CM Master Virtual Axis Command homing
   RUNG wire#powerrail
      Contact( #TRUE )
      Coil( "Unit1.Em3.ControlNodes".cm.Interlock.masterVirtualAxis.source.homing )
   END_RUNG
   RUNG wire#powerrail
      I_Contact( "Unit1.Em3.ControlNodes".webGuid."step".action[151] )
      Not()
      Coil( "Unit1.Em3.ControlNodes".cmMasterVirtualAxis.commands.homing )
   END_RUNG
   // the same network as SCL:
   "Unit1.Em3.ControlNodes".cm.Interlock.masterVirtualAxis.source.homing := #TRUE;
   "Unit1.Em3.ControlNodes".cmMasterVirtualAxis.commands.homing := NOT (NOT "Unit1.Em3.ControlNodes".webGuid."step".action[151]);
END_REGION

REGION Network 38: CM Master Virtual Axis Command posRelative
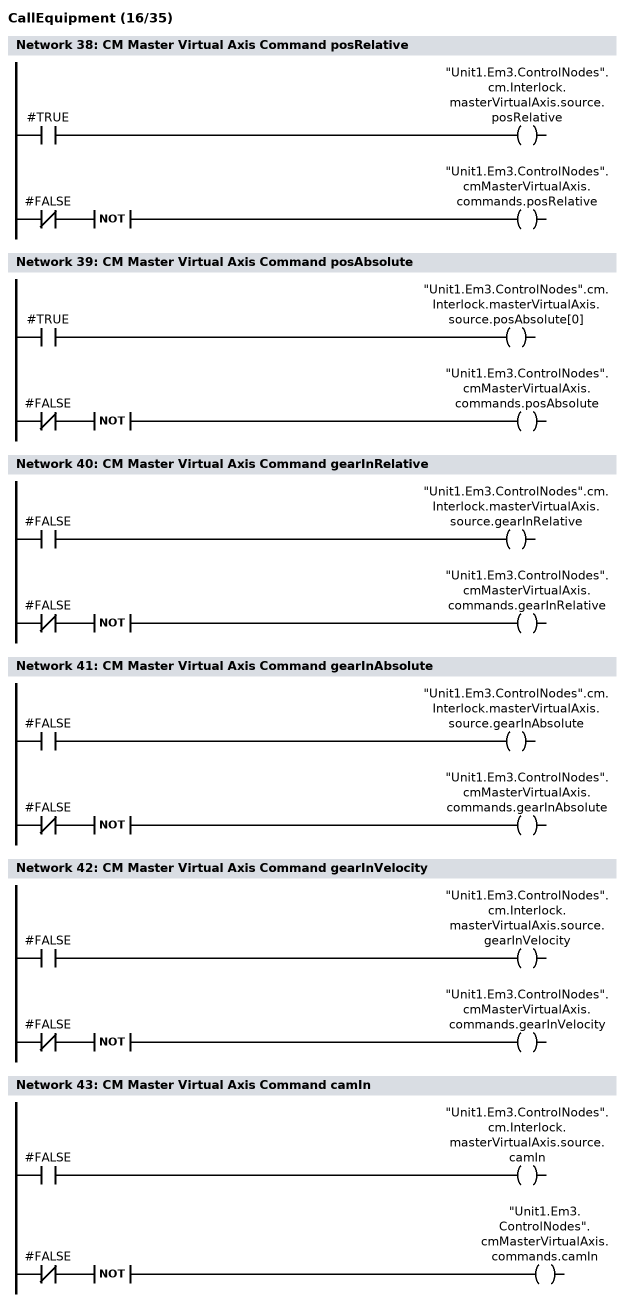
   RUNG wire#powerrail
      Contact( #TRUE )
      Coil( "Unit1.Em3.ControlNodes".cm.Interlock.masterVirtualAxis.source.posRelative )
   END_RUNG
   RUNG wire#powerrail
      I_Contact( #FALSE )
      Not()
      Coil( "Unit1.Em3.ControlNodes".cmMasterVirtualAxis.commands.posRelative )
   END_RUNG
   // the same network as SCL:
   "Unit1.Em3.ControlNodes".cm.Interlock.masterVirtualAxis.source.posRelative := #TRUE;
   "Unit1.Em3.ControlNodes".cmMasterVirtualAxis.commands.posRelative := NOT (NOT #FALSE);
END_REGION

REGION Network 39: CM Master Virtual Axis Command posAbsolute
   RUNG wire#powerrail
      Contact( #TRUE )
      Coil( "Unit1.Em3.ControlNodes".cm.Interlock.masterVirtualAxis.source.posAbsolute[0] )
   END_RUNG
   RUNG wire#powerrail
      I_Contact( #FALSE )
      Not()
      Coil( "Unit1.Em3.ControlNodes".cmMasterVirtualAxis.commands.posAbsolute )
   END_RUNG
   // the same network as SCL:
   "Unit1.Em3.ControlNodes".cm.Interlock.masterVirtualAxis.source.posAbsolute[0] := #TRUE;
   "Unit1.Em3.ControlNodes".cmMasterVirtualAxis.commands.posAbsolute := NOT (NOT #FALSE);
END_REGION

REGION Network 40: CM Master Virtual Axis Command gearInRelative
   RUNG wire#powerrail
      Contact( #FALSE )
      Coil( "Unit1.Em3.ControlNodes".cm.Interlock.masterVirtualAxis.source.gearInRelative )
   END_RUNG
   RUNG wire#powerrail
      I_Contact( #FALSE )
      Not()
      Coil( "Unit1.Em3.ControlNodes".cmMasterVirtualAxis.commands.gearInRelative )
   END_RUNG
   // the same network as SCL:
   "Unit1.Em3.ControlNodes".cm.Interlock.masterVirtualAxis.source.gearInRelative := #FALSE;
   "Unit1.Em3.ControlNodes".cmMasterVirtualAxis.commands.gearInRelative := NOT (NOT #FALSE);
END_REGION

REGION Network 41: CM Master Virtual Axis Command gearInAbsolute
   RUNG wire#powerrail
      Contact( #FALSE )
      Coil( "Unit1.Em3.ControlNodes".cm.Interlock.masterVirtualAxis.source.gearInAbsolute )
   END_RUNG
   RUNG wire#powerrail
      I_Contact( #FALSE )
      Not()
      Coil( "Unit1.Em3.ControlNodes".cmMasterVirtualAxis.commands.gearInAbsolute )
   END_RUNG
   // the same network as SCL:
   "Unit1.Em3.ControlNodes".cm.Interlock.masterVirtualAxis.source.gearInAbsolute := #FALSE;
   "Unit1.Em3.ControlNodes".cmMasterVirtualAxis.commands.gearInAbsolute := NOT (NOT #FALSE);
END_REGION

REGION Network 42: CM Master Virtual Axis Command gearInVelocity
   RUNG wire#powerrail
      Contact( #FALSE )
      Coil( "Unit1.Em3.ControlNodes".cm.Interlock.masterVirtualAxis.source.gearInVelocity )
   END_RUNG
   RUNG wire#powerrail
      I_Contact( #FALSE )
      Not()
      Coil( "Unit1.Em3.ControlNodes".cmMasterVirtualAxis.commands.gearInVelocity )
   END_RUNG
   // the same network as SCL:
   "Unit1.Em3.ControlNodes".cm.Interlock.masterVirtualAxis.source.gearInVelocity := #FALSE;
   "Unit1.Em3.ControlNodes".cmMasterVirtualAxis.commands.gearInVelocity := NOT (NOT #FALSE);
END_REGION

REGION Network 43: CM Master Virtual Axis Command camIn
   RUNG wire#powerrail
      Contact( #FALSE )
      Coil( "Unit1.Em3.ControlNodes".cm.Interlock.masterVirtualAxis.source.camIn )
   END_RUNG
   RUNG wire#powerrail
      I_Contact( #FALSE )
      Not()
      Coil( "Unit1.Em3.ControlNodes".cmMasterVirtualAxis.commands.camIn )
   END_RUNG
   // the same network as SCL:
   "Unit1.Em3.ControlNodes".cm.Interlock.masterVirtualAxis.source.camIn := #FALSE;
   "Unit1.Em3.ControlNodes".cmMasterVirtualAxis.commands.camIn := NOT (NOT #FALSE);
END_REGION

REGION Network 44: CM Master Virtual Axis Command gearOutCamOut
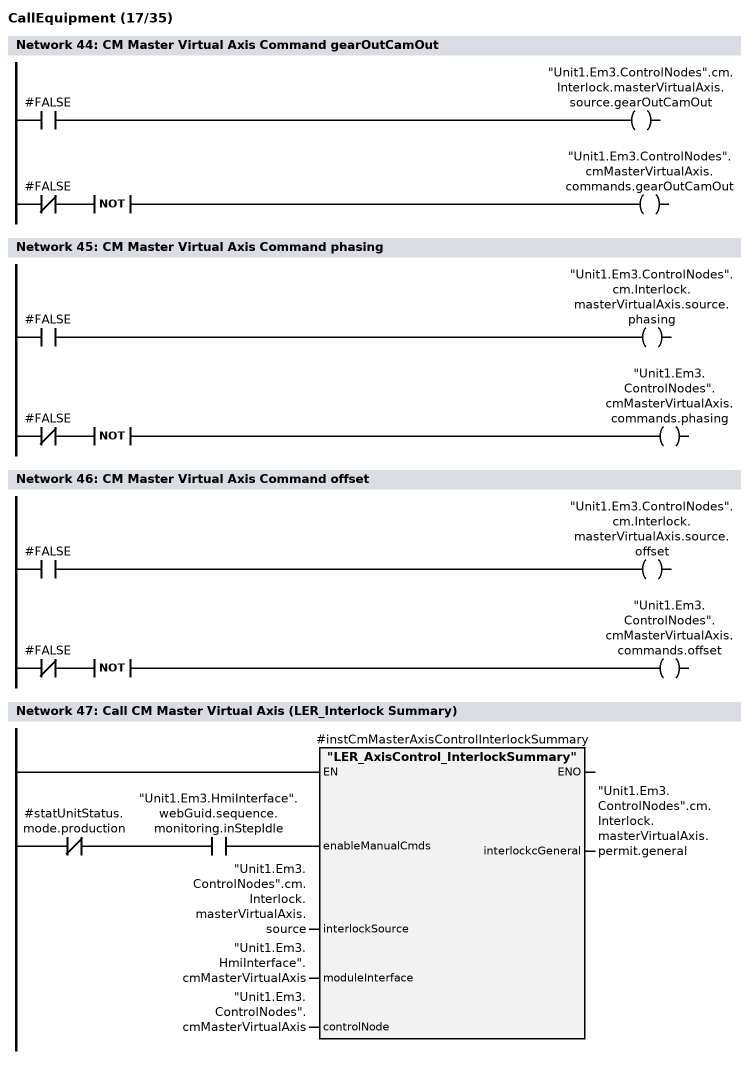
   RUNG wire#powerrail
      Contact( #FALSE )
      Coil( "Unit1.Em3.ControlNodes".cm.Interlock.masterVirtualAxis.source.gearOutCamOut )
   END_RUNG
   RUNG wire#powerrail
      I_Contact( #FALSE )
      Not()
      Coil( "Unit1.Em3.ControlNodes".cmMasterVirtualAxis.commands.gearOutCamOut )
   END_RUNG
   // the same network as SCL:
   "Unit1.Em3.ControlNodes".cm.Interlock.masterVirtualAxis.source.gearOutCamOut := #FALSE;
   "Unit1.Em3.ControlNodes".cmMasterVirtualAxis.commands.gearOutCamOut := NOT (NOT #FALSE);
END_REGION

REGION Network 45: CM Master Virtual Axis Command phasing
   RUNG wire#powerrail
      Contact( #FALSE )
      Coil( "Unit1.Em3.ControlNodes".cm.Interlock.masterVirtualAxis.source.phasing )
   END_RUNG
   RUNG wire#powerrail
      I_Contact( #FALSE )
      Not()
      Coil( "Unit1.Em3.ControlNodes".cmMasterVirtualAxis.commands.phasing )
   END_RUNG
   // the same network as SCL:
   "Unit1.Em3.ControlNodes".cm.Interlock.masterVirtualAxis.source.phasing := #FALSE;
   "Unit1.Em3.ControlNodes".cmMasterVirtualAxis.commands.phasing := NOT (NOT #FALSE);
END_REGION

REGION Network 46: CM Master Virtual Axis Command offset
   RUNG wire#powerrail
      Contact( #FALSE )
      Coil( "Unit1.Em3.ControlNodes".cm.Interlock.masterVirtualAxis.source.offset )
   END_RUNG
   RUNG wire#powerrail
      I_Contact( #FALSE )
      Not()
      Coil( "Unit1.Em3.ControlNodes".cmMasterVirtualAxis.commands.offset )
   END_RUNG
   // the same network as SCL:
   "Unit1.Em3.ControlNodes".cm.Interlock.masterVirtualAxis.source.offset := #FALSE;
   "Unit1.Em3.ControlNodes".cmMasterVirtualAxis.commands.offset := NOT (NOT #FALSE);
END_REGION

